# B&R Automation Studio project Parker_BMM_ST_V5_3147_V12 (part 18)

#### cur_save.c
```c
/********************************************************************
 * COPYRIGHT --  B&R CHINA
 ********************************************************************
 * Program: cur_save
 * File: cur_save.c
 * Author: lijianjun
 * Created: March 06, 2013
 ********************************************************************
 * Implementation of program cur_save --- thick profile curve data save/load
 ********************************************************************/

#include <bur/plctypes.h>
#include <string.h>

#ifdef _DEFAULT_INCLUDES
#include <AsDefault.h>
#endif

/***********************************************************************************
**                            Include user files								  **
***********************************************************************************/
#include "draw.h"
#include "recipe.h"
#include "keyap2100.h"
#include "pic_id.h"

/***********************************************************************************
** 					 	       Macro Define								          **
***********************************************************************************/
#define  S$CURVE_NUM	5

#define S$STEP_INIT_OK  10000

#define S$STEP_IDLE     100
#define S$STEP_READ     1000
#define S$STEP_WRITE    2000

#define S$STEP_ERROR	   30000

#define S$WAIT_COMMAND			   0

#define S$ROOT_DISK_SAVE		   100
#define S$ROOT_DISK_LOAD		   200
#define S$ROOT_DISK_CLEAR		   500

#define S$USB_SINGLE_OPEN_SAVE	1000
#define S$USB_SINGLE_CREATE		1100
#define S$USB_SINGLE_WRITE		   1300

#define S$USB_SINGLE_OPEN_LOAD	2000
#define S$USB_SINGLE_READ_MEM	   2100
#define S$USB_SINGLE_READ			2200

#define S$USB_SINGLE_CLOSE		   3000

#define S$USB_ALL_OPEN_SAVE	   11000
#define S$USB_ALL_CREATE		   11100
#define S$USB_ALL_MEM_ALLOC	   11200
#define S$USB_ALL_MEM_GET	      11300
#define S$USB_ALL_WRITE		      11400
#define S$USB_ALL_MEM_FREE		   11500

#define S$USB_ALL_OPEN_LOAD	   12000
#define S$USB_ALL_ALLOC_MEM	   12100
#define S$USB_ALL_READ			   12200
#define S$USB_ALL_READ_WRITE	   12300
#define S$USB_ALL_FREE_MEM  	   12400

#define S$USB_ALL_CLOSE		      13000

#define S$ERROR_STEP			      40000
/**********************************************************************************
**                          Function Declarations								 **
**********************************************************************************/
void changeCurve(USINT *enable);
void newCurve();
void writeData(UINT Index);
void readData(UINT Index);
void initCurve(unsigned short length);
/**********************************************************************************
**     	        		I N I T U P  O F   T H E   T A S K 		 				 **
**********************************************************************************/
_INIT  void init(void)
{
	strcpy(fileSingleName, "curve.usb");		/* file single name */
	strcpy(fileAllName, "curveAll.usb");		/* file all name */

	strcpy(DataObjOperate.ModName,"recCurve");
	strcpy(DataObjOperate.Status,"");
	DataObjOperate.InitStep = 100;
}/*end of INIT*/

/**********************************************************************************
**        			C Y C L I C   P A R T   O F   T H E   T A S K  				 **
**********************************************************************************/
_CYCLIC void cyc(void)
{
	/*  配方名字及数据初始化  */
	switch(DataObjOperate.InitStep)
	{
		case 100:
			/* Initialize info structure */
			DataObjOperate.Ident = 0;
			DatObj_Info.enable	= 1;
			DatObj_Info.pName	   = (UDINT)DataObjOperate.ModName;

			/* Call  FUB  */
			DatObjInfo(&DatObj_Info);

			if(doERR_MODULNOTFOUND == DatObj_Info.status)
			{
				DatObj_Info.enable = 0;
				DataObjOperate.InitStep = 200;
			}
			else if(0 == DatObj_Info.status)
			{
				DatObj_Info.enable = 0;
				DataObjOperate.Ident = DatObj_Info.ident;
				DataObjOperate.InitStep  = 500;
			}
			else if (DatObj_Info.status != ERR_FUB_BUSY)
			{
				DatObj_Info.enable = 0;
				DataObjOperate.InitStep = 40000;
			}
			break;

		case 200:
			/* Initialize create structure */
			DatObj_Create.enable = 1;
			DatObj_Create.grp	 	= 0;
			DatObj_Create.pName 	= (UDINT)DataObjOperate.ModName;
			DatObj_Create.len 	= sizeof(curveData)*(S$NUM_RECIPE + 1);
				DatObj_Create.MemType  = doUSRROM;
			DatObj_Create.Option   = 0;
			DatObj_Create.pCpyData = 0;

			/* Call FUB */
			DatObjCreate(&DatObj_Create);

			if(0 == DatObj_Create.status)
			{
				DataObjOperate.Ident = DatObj_Create.ident;
				DataObjOperate.InitStep = 300;
			}
			break;

		case 300:
			counter = 0;
			initCurve(S$THICK_INIT_LENGTH);
				DataObjOperate.InitStep = 350;
			break;

		case 350:
			status_tmpalloc = TMP_alloc(sizeof(curveData) * (S$NUM_RECIPE + 1), (void*)&pCurveData);
				if(0 == status_tmpalloc)
			{
				for(i=0;i<(S$NUM_RECIPE+1) * S$CURVE_NUM;i++)
					{
					((curveData_typ *)pCurveData)[i] = curveData[0];
				}
				DataObjOperate.InitStep = 380;
			}
			else
			{
				DataObjOperate.InitStep = 40001;
			}
			break;

		case 380:
			DatObj_Write.enable  = 1;
			DatObj_Write.ident 	= DataObjOperate.Ident;
			DatObj_Write.Offset  = 0;
			DatObj_Write.pSource = (UDINT)pCurveData;
			DatObj_Write.len 	   = sizeof(curveData) * (S$NUM_RECIPE + 1);

				/* Call FUB */
				DatObjWrite(&DatObj_Write);

			if(0 == DatObj_Write.status )
			{
				DataObjOperate.InitStep = 400;
			}
			break;

		case 400:
			status_tmpfree = TMP_free(sizeof(curveData) * (S$NUM_RECIPE + 1), (void*)pCurveData);
				if(0 == status_tmpfree)
			{
				readData(curveIndex);
				DataObjOperate.InitStep = 700;
			}
			else
			{
				DataObjOperate.InitStep = 40002;
			}
			break;

		case 500:
			if(1 == gRecipeOperate.NameOk)
			{
				DataObjOperate.InitStep = 600;
			}
			break;

		case 600:
			/* Initialize read structure */
			DatObj_Read.enable 		 = 1;
			DatObj_Read.ident 		 = DataObjOperate.Ident;
			DatObj_Read.Offset 		 = sizeof(curveData) * S$NUM_RECIPE;
			DatObj_Read.pDestination = (UDINT) &curveData;
			DatObj_Read.len 		    = sizeof (curveData);

			/* Call FUB */
			DatObjRead(&DatObj_Read);
			if (curveData[0].usedIndex < S$CURVE_NUM )
				{
				curveIndex = curveData[0].usedIndex;
			}
			else
			{
				curveIndex	= S$CURVE_NUM - 1;
			}

			readData(curveIndex);

			if(0 == DatObj_Read.status)
			{
				DataObjOperate.InitStep = 700;
			}
			else
			{
				DataObjOperate.InitStep = S$STEP_ERROR;
			}
			break;

		case 700:       /*   recipe data  ok*/
			gRecipeOperate.CurveOk  = 1;
			strcpy(DataObjOperate.Status,"curvedata init ok !");
			DataObjOperate.Step     = S$STEP_IDLE;
			DataObjOperate.InitStep = S$STEP_INIT_OK;
			break;

		case S$STEP_INIT_OK:
				break;

		case S$STEP_ERROR:
				break;

		default:
			break;
	}/* switch(DataObjOperate.InitStep) */

	if((0 == DataObjOperate.Ident)||(DataObjOperate.InitStep != S$STEP_INIT_OK ))
		{
		gRecipeOperate.CurveUSBSave = 0;
		gRecipeOperate.CurveUSBLoad = 0;
		curveIndexOld = curveIndex;
		return;
	}

	/* ----------------- Step machine control ----------------- */
	switch (DataObjOperate.Step)
	{
		case S$WAIT_COMMAND:
				gRecipeOperate.usbCurveOk = 1;
			if(1 == gRecipeOperate.CurveSave)
			{
				gRecipeOperate.CurveSave = 0;
				indexRecipe = S$NUM_RECIPE;			/*  current recipe in data module-index = S$NUM_RECIPE */
				DataObjOperate.Step = S$ROOT_DISK_SAVE;
			}/* else if(1 == gRecipeOperate.CurveSave) */
			else if(1 == gRecipeOperate.CurveLoad)
			{
				gRecipeOperate.CurveLoad = 0;
				indexRecipe = S$NUM_RECIPE;			/*  current recipe in data module-index = S$NUM_RECIPE */
				DataObjOperate.Step = S$ROOT_DISK_LOAD;
			}/* else if(1 == gRecipeOperate.CurveSave) */
			else if(1 == gRecipeOperate.CurveRecipeSave)
			{
				gRecipeOperate.CurveRecipeSave = 0;
				indexRecipe = gRecipeOperate.Index % S$NUM_RECIPE;
				DataObjOperate.Step = S$ROOT_DISK_SAVE;
			}/* else if(1 == gRecipeOperate.CurveSave) */
			else if(1 == gRecipeOperate.CurveRecipeLoad)
			{
				gRecipeOperate.CurveRecipeLoad = 0;
				indexRecipe = gRecipeOperate.Index % S$NUM_RECIPE;
				DataObjOperate.Step = S$ROOT_DISK_LOAD;
				gRecipeOperate.CurveSave = 1;		/*  read from recipe then write to current recipe(S$NUM_RECIPE) in data module */
			}/* else if(1 == gRecipeOperate.CurveSave) */
			else if(1 == gRecipeOperate.CurveUSBSave)
			{
				gRecipeOperate.usbCurveOk = 0;
				gRecipeOperate.CurveUSBSave = 0;
				DataObjOperate.Step = S$USB_SINGLE_OPEN_SAVE;
			}/* else if(1 == gRecipeOperate.CurveUSBSave) */
			else if(1 == gRecipeOperate.CurveUSBLoad)
			{
				gRecipeOperate.usbCurveOk = 0;
				gRecipeOperate.CurveUSBLoad = 0;
				DataObjOperate.Step = S$USB_SINGLE_OPEN_LOAD;
				gRecipeOperate.CurveSave = 1;		/*  read from USB then write to current recipe(S$NUM_RECIPE) in data module */
			}/* else if(1 == gRecipeOperate.CurveUSBLoad) */
			else if(1 == gRecipeOperate.CurveUSBLoadAll)
			{
				gRecipeOperate.usbCurveOk = 0;
				gRecipeOperate.CurveUSBLoadAll = 0;
				DataObjOperate.Step = S$USB_ALL_OPEN_LOAD;
			}
			else if(1 == gRecipeOperate.CurveUSBSaveAll)
			{
				gRecipeOperate.usbCurveOk = 0;
				gRecipeOperate.CurveUSBSaveAll = 0;
				DataObjOperate.Step = S$USB_ALL_OPEN_SAVE;
			}
			break;

		/* ---------------- Save to root disk ---------------- */
		case S$ROOT_DISK_SAVE:
				curveData[0].usedIndex = curveIndex;
			writeData(curveIndex);
			/* Initialize write structure */
			DatObj_Write.enable 	= 1;
			DatObj_Write.ident 	= DataObjOperate.Ident;
			DatObj_Write.Offset 	= sizeof(curveData)*indexRecipe;
			DatObj_Write.pSource = (UDINT)&curveData;
			DatObj_Write.len 	   = sizeof(curveData);

			/* Call FUB */
			DatObjWrite(&DatObj_Write);

			if(DatObj_Write.status == 0)
			{
				strcpy(DataObjOperate.Status,"curvedata write ok !");
			}
			else
			{
				strcpy(DataObjOperate.Status,"curvedata write false !");
			}

			DataObjOperate.Step = S$WAIT_COMMAND;
			break;

		/* ---------------- Load from root disk ---------------- */
		case S$ROOT_DISK_LOAD:
				/* Initialize read structure */
				DatObj_Read.enable 		  = 1;
			DatObj_Read.ident 		  = DataObjOperate.Ident;
			DatObj_Read.Offset 		  = sizeof(curveData)*indexRecipe;
			DatObj_Read.pDestination  = (UDINT)&curveData;
			DatObj_Read.len 		     = sizeof(curveData);

			/* Call FUB */
			DatObjRead(&DatObj_Read);

			if(DatObj_Read.status == 0)
			{
				strcpy(DataObjOperate.Status,"curvedata read ok !");
			}
			else
			{
				strcpy(DataObjOperate.Status,"curvedata read false !");
			}

			if (curveData[0].usedIndex < S$CURVE_NUM)
				{
				curveIndex = curveData[0].usedIndex;
			}
			else
			{
				curveIndex	= S$CURVE_NUM - 1;
			}

			readData(curveIndex);

			DataObjOperate.Step = S$WAIT_COMMAND;
			break;

		/* --------------------------------------------------------------- */
		/* ---------------- Save Single curve to usb disk ---------------- */
		/* --------------------------------------------------------------- */
		case S$USB_SINGLE_OPEN_SAVE:			/* file OPEN for save  */
				FileOpen_0.enable  = 1;
			FileOpen_0.pDevice = (UDINT)&gRecipeOperate.deviceNameUSB;
			FileOpen_0.pFile   = (UDINT)&fileSingleName;
			FileOpen_0.mode    = fiREAD_WRITE;

			/* Call FUB */
			FileOpen(&FileOpen_0);

			if(fiERR_FILE_NOT_FOUND == FileOpen_0.status)/* no file   */
			{
				FileOpen_0.enable  = 0;
				DataObjOperate.Step = S$USB_SINGLE_CREATE;
			}
			else
			{
				if(ERR_OK == FileOpen_0.status)			/* file exist */
				{
					FileOpen_0.enable  = 0;
					if(FileOpen_0.filelen == sizeof(curveData))
					{
						DataObjOperate.IdentUSB = FileOpen_0.ident;
						DataObjOperate.Step = S$USB_SINGLE_WRITE;
					}
					else
					{
						gImply.CurveUSB_Length = 1;
						DataObjOperate.Step = S$USB_SINGLE_CLOSE;
					}
				}
				else if (FileOpen_0.status != ERR_FUB_BUSY)
				{
					FileOpen_0.enable  = 0;
					gImply.CurveOP_False = 1;
					DataObjOperate.Step = S$ERROR_STEP;
				}
			}
			break;

		case S$USB_SINGLE_CREATE:			/* file not exist, create*/
				FileCreate_0.enable  = 1;
			FileCreate_0.pDevice = (UDINT)&gRecipeOperate.deviceNameUSB;
			FileCreate_0.pFile   = (UDINT)&fileSingleName;

			/* Call FUB */
			FileCreate(&FileCreate_0);

			if(ERR_OK == FileCreate_0.status)		/* ok */
			{
				FileCreate_0.enable = 0;
				DataObjOperate.IdentUSB = FileCreate_0.ident;
				DataObjOperate.Step = S$USB_SINGLE_WRITE;
			}
			else if (FileCreate_0.status != ERR_FUB_BUSY)
			{
				FileCreate_0.enable= 0;
				gImply.CurveOP_False = 1;
				DataObjOperate.Step = S$USB_SINGLE_CLOSE;
			}
			break;

		case S$USB_SINGLE_WRITE:		/* file write */
				FileWrite_0.enable = 1;
			FileWrite_0.ident  = DataObjOperate.IdentUSB;
			FileWrite_0.offset = 0;
			FileWrite_0.pSrc = (UDINT)&curveData;
			FileWrite_0.len  = sizeof(curveData);

			/* Call FUB */
			FileWrite(&FileWrite_0);

			if(ERR_OK == FileWrite_0.status)				/* ok */
			{
				FileWrite_0.enable = 0;
				gImply.CurveOP_OK = 1;
				DataObjOperate.Step = S$USB_SINGLE_CLOSE;
			}
			else if (FileWrite_0.status != ERR_FUB_BUSY)
			{
				FileWrite_0.enable = 0;
				gImply.CurveOP_False = 1;
				DataObjOperate.Step = S$USB_SINGLE_CLOSE;
			}
			break;

		/* ----------------------------------------------------------------- */
		/* ---------------- Load single curve from USB disk ---------------- */
		/* ----------------------------------------------------------------- */
		case S$USB_SINGLE_OPEN_LOAD:			/* file OPEN  for load  */
				FileOpen_0.enable  = 1;
			FileOpen_0.pDevice = (UDINT)&gRecipeOperate.deviceNameUSB;
			FileOpen_0.pFile   = (UDINT)&fileSingleName;
			FileOpen_0.mode    = fiREAD_WRITE;

			/* Call FUB */
			FileOpen(&FileOpen_0);

			if(fiERR_FILE_NOT_FOUND == FileOpen_0.status)	/* no file   */
			{
				FileOpen_0.enable  = 0;
				gImply.FixUSB_NoFile = 1;
				DataObjOperate.Step = S$WAIT_COMMAND;
			}
			else
			{
				if(ERR_OK == FileOpen_0.status)				/* file exist */
				{
					FileOpen_0.enable = 0;
					if(FileOpen_0.filelen == sizeof(curveData))
					{
						DataObjOperate.IdentUSB = FileOpen_0.ident;
						DataObjOperate.Step = S$USB_SINGLE_READ;
					}
					else
					{
						gImply.CurveUSB_Length = 1;
						DataObjOperate.Step = S$USB_SINGLE_CLOSE;
					}
				}
				else if (FileOpen_0.status != ERR_FUB_BUSY)
				{
					FileOpen_0.enable = 0;
					gImply.CurveOP_False = 1;
					DataObjOperate.Step = S$ERROR_STEP;
				}
			}
			break;

		case S$USB_SINGLE_READ:			/* file single read  */
				FileRead_0.enable = 1;
			FileRead_0.ident  = DataObjOperate.IdentUSB;
			FileRead_0.offset = 0;
			FileRead_0.pDest  = (UDINT)&curveData;
			FileRead_0.len    = sizeof(curveData);

			/* Call FUB */
			FileRead(&FileRead_0);

			if(ERR_OK == FileRead_0.status)	/* ok */
			{
				FileRead_0.enable = 0;
				gImply.CurveOP_OK = 1;
				if (curveData[0].usedIndex < S$CURVE_NUM)
					{
					curveIndex = curveData[0].usedIndex;
				}
				else
				{
					curveIndex	= S$CURVE_NUM - 1;
				}

				readData(curveIndex);

				gRecipeOperate.CurveSave = 1;		/*  read from USB then write to current recipe(S$NUM_RECIPE) in data module */
				DataObjOperate.Step = S$USB_SINGLE_CLOSE;
			}
			else if (FileRead_0.status != ERR_FUB_BUSY)
			{
				FileRead_0.enable = 0;
				gImply.CurveOP_False = 1;
				DataObjOperate.Step = S$USB_SINGLE_CLOSE;
			}
			break;

		/* ------------------------------------------------------- */
		/* ---------------- Close USB file device ---------------- */
		/* ------------------------------------------------------- */
		case S$USB_SINGLE_CLOSE:			/* file close*/
				FileClose_0.enable = 1;
			FileClose_0.ident  = DataObjOperate.IdentUSB;

			/* Call FBK */
			FileClose(&FileClose_0);

			if(ERR_OK == FileClose_0.status)	/* ok */
			{
				FileClose_0.enable = 0;
				DataObjOperate.Step = S$WAIT_COMMAND;
			}
			else if (FileClose_0.status != ERR_FUB_BUSY)
			{
				FileClose_0.enable = 0;
				DataObjOperate.Step = S$ERROR_STEP;
			}
			break;

		/* ------------------------------------------------------ */
		/* ---------------- All Save to usb disk ---------------- */
		/* ------------------------------------------------------ */
		case S$USB_ALL_OPEN_SAVE:			/* file OPEN for save  */
				FileOpen_0.enable  = 1;
			FileOpen_0.pDevice = (UDINT)&gRecipeOperate.deviceNameUSB;
			FileOpen_0.pFile   = (UDINT)&fileAllName;
			FileOpen_0.mode    = fiREAD_WRITE;

			/* Call FUB */
			FileOpen(&FileOpen_0);

			if(fiERR_FILE_NOT_FOUND == FileOpen_0.status)/* no file   */
			{
				FileOpen_0.enable   = 0;
				DataObjOperate.Step = S$USB_ALL_CREATE;
			}
			else
			{
				if(ERR_OK == FileOpen_0.status)			/* file exist */
				{
					FileOpen_0.enable  = 0;
					if(FileOpen_0.filelen == sizeof(curveData)*(S$NUM_RECIPE + 1))
						{
						DataObjOperate.IdentAllUSB = FileOpen_0.ident;
						DataObjOperate.Step = S$USB_ALL_MEM_ALLOC;
					}
					else
					{
						gImply.CurveUSB_Length = 1;
						DataObjOperate.Step = S$USB_ALL_CLOSE;
					}
				}
				else if (FileOpen_0.status != ERR_FUB_BUSY)
				{
					FileOpen_0.enable  = 0;
					gImply.CurveOP_False = 1;
					DataObjOperate.Step = S$ERROR_STEP;
				}
			}
			break;

		case S$USB_ALL_CREATE:			/* file not exist, create*/
				FileCreate_0.enable  = 1;
			FileCreate_0.pDevice = (UDINT)&gRecipeOperate.deviceNameUSB;
			FileCreate_0.pFile   = (UDINT)&fileAllName;

			/* Call FUB */
			FileCreate(&FileCreate_0);

			if(ERR_OK == FileCreate_0.status)		/* ok */
			{
				FileCreate_0.enable = 0;
				DataObjOperate.IdentAllUSB = FileCreate_0.ident;
				DataObjOperate.Step = S$USB_ALL_MEM_ALLOC;
			}
			else if (FileCreate_0.status != ERR_FUB_BUSY)
			{
				FileCreate_0.enable = 0;
				gImply.CurveOP_False = 1;
				DataObjOperate.Step = S$USB_ALL_CLOSE;
			}
			break;

		case S$USB_ALL_MEM_ALLOC:	/* file request All memory */
				status_tmpalloc = TMP_alloc(sizeof(curveData)*(S$NUM_RECIPE + 1), (void*)&pCurveData);
				if(0 == status_tmpalloc)
			{
				memset((void *)pCurveData,0,sizeof(curveData)*(S$NUM_RECIPE + 1));
					DataObjOperate.Step = S$USB_ALL_MEM_GET;
			}
			else
			{
				gImply.CurveOP_False = 1;
				DataObjOperate.Step = S$USB_ALL_CLOSE;
			}
			break;

		case S$USB_ALL_MEM_GET:
				DatObj_Read.enable = 1;
			DatObj_Read.ident  = DataObjOperate.Ident;
			DatObj_Read.Offset = 0;
			DatObj_Read.pDestination = (UDINT)pCurveData;
			DatObj_Read.len = sizeof(curveData)*(S$NUM_RECIPE + 1);

				/* Call FUB */
				DatObjRead(&DatObj_Read);
			if(0 == DatObj_Read.status)
			{
				DatObj_Read.enable = 0;
				DataObjOperate.Step = S$USB_ALL_WRITE;
			}
			else if (DatObj_Read.status != ERR_FUB_BUSY)
			{
				DatObj_Read.enable = 0;
				gImply.CurveOP_False = 1;
				DataObjOperate.Step = S$USB_ALL_MEM_FREE;
			}
			break;

		case S$USB_ALL_WRITE:		/* file single write */
				FileWrite_0.enable = 1;
			FileWrite_0.ident  = DataObjOperate.IdentAllUSB;
			FileWrite_0.offset = 0;
			FileWrite_0.pSrc = (UDINT)pCurveData;
			FileWrite_0.len  = sizeof(curveData)*(S$NUM_RECIPE + 1);

				/* Call FUB */
				FileWrite(&FileWrite_0);

			if(ERR_OK == FileWrite_0.status)				/* ok */
			{
				FileWrite_0.enable = 0;
				gImply.CurveOP_OK = 1;
				DataObjOperate.Step = S$USB_ALL_MEM_FREE;
			}
			else if (FileWrite_0.status != ERR_FUB_BUSY)
			{
				FileWrite_0.enable = 0;
				gImply.CurveOP_False = 1;
				DataObjOperate.Step = S$USB_ALL_MEM_FREE;
			}
			break;

		case S$USB_ALL_MEM_FREE:
				status_tmpfree = TMP_free(sizeof(curveData)*(S$NUM_RECIPE + 1), (void*)pCurveData);
				if(0 == status_tmpfree)
			{
				DataObjOperate.Step = S$USB_ALL_CLOSE;
			}
			else
			{
				DataObjOperate.Step = S$USB_ALL_CLOSE;
			}
			break;

		/* ----------------------------------------------------------- */
		/* ----------------  All Load from USB disk   ---------------- */
		/* ----------------------------------------------------------- */
		case S$USB_ALL_OPEN_LOAD:			/* file OPEN  for load  */
				FileOpen_0.enable  = 1;
			FileOpen_0.pDevice = (UDINT)&gRecipeOperate.deviceNameUSB;
			FileOpen_0.pFile   = (UDINT)&fileAllName;
			FileOpen_0.mode    = fiREAD_WRITE;

			/* Call FUB */
			FileOpen(&FileOpen_0);

			if(fiERR_FILE_NOT_FOUND == FileOpen_0.status)	/* no file   */
			{
				FileOpen_0.enable  = 0;
				gImply.CurveUSB_NoFile = 1;
				DataObjOperate.Step = S$WAIT_COMMAND;
			}
			else
			{
				if(ERR_OK == FileOpen_0.status)				/* file exist */
				{
					FileOpen_0.enable = 0;
					if(FileOpen_0.filelen == sizeof(curveData)*(S$NUM_RECIPE + 1))
						{
						DataObjOperate.IdentAllUSB = FileOpen_0.ident;
						DataObjOperate.Step = S$USB_ALL_ALLOC_MEM;
					}
					else
					{
						gImply.CurveUSB_Length = 1;
						DataObjOperate.Step = S$USB_ALL_CLOSE;
					}
				}
				else if (FileOpen_0.status != ERR_FUB_BUSY)
				{
					FileOpen_0.enable = 0;
					gImply.CurveOP_False = 1;
					DataObjOperate.Step = S$ERROR_STEP;
				}
			}
			break;

		case S$USB_ALL_ALLOC_MEM:			/* file  read request memory */
				status_tmpalloc = TMP_alloc(sizeof(curveData)*(S$NUM_RECIPE + 1), (void*)&pCurveData);
				if(0 == status_tmpalloc)
			{
				DataObjOperate.Step = S$USB_ALL_READ;
			}
			else
			{
				gImply.CurveOP_False = 1;
				DataObjOperate.Step = S$USB_ALL_CLOSE;
			}
			break;

		case S$USB_ALL_READ:			/* file  read  */
				FileRead_0.enable = 1;
			FileRead_0.ident  = DataObjOperate.IdentAllUSB;
			FileRead_0.offset = 0;
			FileRead_0.pDest  = (UDINT)pCurveData;
			FileRead_0.len    = sizeof(curveData)*(S$NUM_RECIPE + 1);

				/* Call FUB */
				FileRead(&FileRead_0);

			if(ERR_OK == FileRead_0.status)	/* ok */
			{
				FileRead_0.enable = 0;
				DataObjOperate.Step = S$USB_ALL_READ_WRITE;
			}
			else if (FileRead_0.status != ERR_FUB_BUSY)
			{
				FileRead_0.enable = 0;
				gImply.CurveOP_False = 1;
				DataObjOperate.Step = S$USB_ALL_FREE_MEM;
			}
			break;

		case S$USB_ALL_READ_WRITE:
				DatObj_Write.enable  = 1;
			DatObj_Write.ident 	 = DataObjOperate.Ident;
			DatObj_Write.Offset  = 0;
			DatObj_Write.pSource = (UDINT)pCurveData;
			DatObj_Write.len 	 = sizeof(curveData)*(S$NUM_RECIPE + 1);

				DatObjWrite(&DatObj_Write);

			if(0 == DatObj_Write.status)
			{
				DatObj_Write.enable  = 0;
				gImply.CurveOP_OK = 1;
				gRecipeOperate.CurveLoad = 1;
				DataObjOperate.Step = S$USB_ALL_FREE_MEM;
			}
			else if (DatObj_Write.status != ERR_FUB_BUSY)
			{
				DatObj_Write.enable  = 0;
				gImply.CurveOP_False = 1;
				DataObjOperate.Step = S$USB_ALL_FREE_MEM;
			}
			break;

		case S$USB_ALL_FREE_MEM:
				status_tmpfree = TMP_free(sizeof(curveData)*(S$NUM_RECIPE + 1), (void*)pCurveData);
				if(0 == status_tmpfree)
			{
				DataObjOperate.Step = S$USB_ALL_CLOSE;
			}
			else
			{
				DataObjOperate.Step = S$USB_ALL_CLOSE;
			}
			break;
		/* ----------------------------------------------------------- */
		/* ---------------- All Close USB file device ---------------- */
		/* ----------------------------------------------------------- */
		case S$USB_ALL_CLOSE:			/* file close*/
				FileClose_0.enable = 1;
			FileClose_0.ident  = DataObjOperate.IdentAllUSB;

			/* Call FBK */
			FileClose(&FileClose_0);

			if(ERR_OK == FileClose_0.status)	/* ok */
			{
				FileClose_0.enable = 0;
				DataObjOperate.Step = S$WAIT_COMMAND;
			}
			else if (FileClose_0.status != ERR_FUB_BUSY)
			{
				FileClose_0.enable = 0;
				DataObjOperate.Step = S$ERROR_STEP;
			}
			break;

		case S$ERROR_STEP:
				DataObjOperate.Step = S$WAIT_COMMAND;
			break;
	}/* switch (DataObjOperate.Step) */

	if(1 == bCurveIndexChgBtn)
	{
		bCurveIndexChgBtn = 0;
		curveIndex = curveIndex + 1;
		curveIndex = curveIndex % 5;
	}

	if(curveIndex != curveIndexOld)
	{
		ChangeEnable = 1;
		changeCurve(&ChangeEnable);
		bCurveIndexChange = 1;
	}
	curveIndexOld = curveIndex;

}/*end of CYCLIC*/

/**************************************************************************************
**        				FUNCTION  REALIZE				   							 **
**************************************************************************************/
void changeCurve(USINT *enable)
{

	if (1 == *enable)
	{
		writeData(curveIndexOld);

		/*curveIndex = curveIndex + 1;*/

		curveIndex = curveIndex % S$CURVE_NUM;

		if (curveData[curveIndex].CurveNode[S$THICK_MAX].v3.y == 0)
			{
			newCurve();
		}
		else
		{
			readData(curveIndex);
		}

		*enable = 0;
	}
}

void newCurve()
{
	memset(SetPos,0,sizeof(SetPos));
	memset(CurveNode,0,sizeof(CurveNode));

	for( i = 0; i<= S$THICK_MAX; i++)
		{
		DrawMan.weight = 300;
		SetPos[i].x = DrawMan.weight;
		SetPos[i].y = i;
	}

	DrawMan.oldWeight 			=  DrawMan.weight;
	DrawMan.v1 						=  (DrawMan.weight) + 1;
	DrawMan.v2 						=  (DrawMan.weight) + 1;
	DrawMan.v03 					=  0;
	DrawMan.currentNode  		=  S$THICK_MAX;
	DrawMan.currentPoint 		=  0;
	DrawMan.flagLineFocus 		=  0;
	CurveNode[0].former    	=  S$THICK_MAX;
	CurveNode[0].next    		=  S$THICK_MAX;
	CurveNode[0].v3.x    		=  DrawMan.weight;
	CurveNode[0].v3.y    		=  0;
	CurveNode[0].flagNode  		=  1;

	CurveNode[S$THICK_MAX].former 	= 0;
	CurveNode[S$THICK_MAX].next   	= 0;
	CurveNode[S$THICK_MAX].v0.x   	= DrawMan.weight;
	CurveNode[S$THICK_MAX].v0.y   	= 0;
	CurveNode[S$THICK_MAX].v3.x   	= DrawMan.weight;
	CurveNode[S$THICK_MAX].v3.y   	= S$THICK_MAX;

	CurveNode[S$THICK_MAX].v1.x   	= (DrawMan.weight) + 1;
	CurveNode[S$THICK_MAX].v1.y   	= CurveNode[S$THICK_MAX].v0.y +
		(CurveNode[S$THICK_MAX].v3.y - CurveNode[S$THICK_MAX].v0.y)*1/
		3 ;
		CurveNode[S$THICK_MAX].v2.x   	= (DrawMan.weight) + 1;
	CurveNode[S$THICK_MAX].v2.y   	= CurveNode[S$THICK_MAX].v0.y +
		(CurveNode[S$THICK_MAX].v3.y - CurveNode[S$THICK_MAX].v0.y)*(S$THICK_V_SCALE -1)/
		S$THICK_V_SCALE;

	CurveNode[S$THICK_MAX].flagNode =  1;

	setColor = 1;
}/*end of function */

void readData(UINT Index)
{
	Index = Index % 5;
	memcpy(CurveNode,curveData[Index].CurveNode,sizeof(CurveNode));
	memcpy(SetPos,curveData[Index].SetPos,sizeof(SetPos));
	DrawMan.weight 	   = 	curveData[Index].weight;
	DrawMan.oldWeight 	=  DrawMan.weight;
	DrawMan.v1 				= 	curveData[Index].v1;
	DrawMan.v2				= 	curveData[Index].v2;
	DrawMan.v03				= 	curveData[Index].v03;
	DrawMan.currentPoint	=	curveData[Index].currentPoint;
	DrawMan.currentNode	=	curveData[Index].currentNode;
	DrawMan.flagLineFocus=	curveData[Index].flagLineFocus;

}/*end of function */

void writeData(UINT Index)
{
	Index = Index % 5;
	memcpy(curveData[Index].CurveNode,CurveNode,sizeof(CurveNode));
	memcpy(curveData[Index].SetPos,SetPos,sizeof(SetPos));
	curveData[Index].weight 			= 	DrawMan.weight;
	curveData[Index].v1 				   = 	DrawMan.v1;
	curveData[Index].v2			      = 	DrawMan.v2;
	curveData[Index].v03				   = 	DrawMan.v03;
	curveData[Index].currentPoint	   =	DrawMan.currentPoint;
	curveData[Index].currentNode	   =	DrawMan.currentNode;
	curveData[Index].flagLineFocus	=	DrawMan.flagLineFocus;

}/*end of function */
void initCurve(unsigned short length)
{
	memset(curveData[0].SetPos,0,sizeof(curveData[0].SetPos));
	memset(curveData[0].CurveNode,0,sizeof(curveData[0].CurveNode));

	for( i = 0; i<= S$THICK_MAX; i++)
		{
		curveData[0].SetPos[i].x = length;
		curveData[0].SetPos[i].y = i;
	}

	curveData[0].weight        =  0;
	curveData[0].v1 	         =  length+1;
	curveData[0].v2		      =  length+1;
	curveData[0].v03	         =  length;
	curveData[0].currentNode   =  S$THICK_MAX;
	curveData[0].currentPoint  =  0;
	curveData[0].flagLineFocus =  0;
	curveData[0].usedIndex     =  0;

	curveData[0].CurveNode[0].former   =  S$THICK_MAX;
	curveData[0].CurveNode[0].next     =  S$THICK_MAX;
	curveData[0].CurveNode[0].v3.x     =  length;
	curveData[0].CurveNode[0].v3.y     =  0;
	curveData[0].CurveNode[0].flagNode  =  1;

	curveData[0].CurveNode[S$THICK_MAX].former 	= 0;
	curveData[0].CurveNode[S$THICK_MAX].next   	= 0;
	curveData[0].CurveNode[S$THICK_MAX].v0.x   	= length;
	curveData[0].CurveNode[S$THICK_MAX].v0.y   	= 0;
	curveData[0].CurveNode[S$THICK_MAX].v3.x   	= length;
	curveData[0].CurveNode[S$THICK_MAX].v3.y   	= S$THICK_MAX;

	curveData[0].CurveNode[S$THICK_MAX].v1.x   	= length+1;
	curveData[0].CurveNode[S$THICK_MAX].v1.y   	= CurveNode[S$THICK_MAX].v0.y +
		(curveData[0].CurveNode[S$THICK_MAX].v3.y - curveData[0].CurveNode[S$THICK_MAX].v0.y)*1/3 ;
		curveData[0].CurveNode[S$THICK_MAX].v2.x   	= length+1;
	curveData[0].CurveNode[S$THICK_MAX].v2.y   	= CurveNode[S$THICK_MAX].v0.y +
		(curveData[0].CurveNode[S$THICK_MAX].v3.y - curveData[0].CurveNode[S$THICK_MAX].v0.y)*2/3;
		curveData[0].CurveNode[S$THICK_MAX].flagNode =  1;

	memcpy(&curveData[1],&curveData[0],sizeof(curveData_typ));
	memcpy(&curveData[2],&curveData[0],sizeof(curveData_typ));
	memcpy(&curveData[3],&curveData[0],sizeof(curveData_typ));
	memcpy(&curveData[4],&curveData[0],sizeof(curveData_typ));
}

/*************************************************************************************/
```

### Program Logical/thickness/cur_cal (ANSIC, version 1.00.0) - profile point value

#### cur_cal.c
```c
/**************************************************************************************
 * COPYRIGHT --  B&R CHINA
 **************************************************************************************
 * Program: cur_cal
 * File: cur_cal.c
 * Author: lijianjun
 * Created: March 06, 2013
 *************************************************************************************
 * Implementation of program cur_cal --- thick profile curve data calculation
 ************************************************************************************/

#include <bur/plctypes.h>
#include <string.h>

#ifdef _DEFAULT_INCLUDES
#include <AsDefault.h>
#endif

/***********************************************************************************
** 					 	           Include user files								          **
***********************************************************************************/
#include "draw.h"

/**********************************************************************************
**                             Function Declarations								      **
**********************************************************************************/
void BesselCal(short nodeNum);

/**********************************************************************************
**     	        		      I N I T U P  O F   T H E   T A S K 		 				   **
**********************************************************************************/
_INIT void init ( void )
{
	calStep = 0;
}

/**********************************************************************************
**        			 C Y C L I C   P A R T   O F   T H E   T A S K  				   **
**********************************************************************************/
_CYCLIC void cyclic ( void )
{
	if (oldV2 != DrawMan.v2   && enable == 0 && calStep == 0)enable = 1;
	if (oldV1 != DrawMan.v1   && enable == 0 && calStep == 0)enable = 1;
	if (oldV03 != DrawMan.v03 && enable == 0 && calStep == 0)enable = 1;

	SetPos[0].x  = CurveNode[0].v3.x;
	SetPos[0].y  = 0;
	SetPos[S$THICK_MAX].x = CurveNode[S$THICK_MAX].v3.x;
	SetPos[S$THICK_MAX].y = S$THICK_MAX;

	BesselCal(DrawMan.currentNode);

}/*end of CYCLIC*/

/**************************************************************************************
**        				          FUNCTION  REALIZE				   							 **
**************************************************************************************/
void BesselCal(short nodeNum)
{
	switch (calStep)
	{
		case 0:
			if (1 == enable)
			{
				p0 = &CurveNode[nodeNum];
				p1 = &CurveNode[CurveNode[nodeNum].next];

				v1  = DrawMan.v1;
				v2  = DrawMan.v2;
				v03 = DrawMan.v03;
				if ((p0->v3.y - p0->v0.y) != 0) interval0	= 1/(float)(p0->v3.y - p0->v0.y);
				if ((p1->v3.y - p1->v0.y) != 0) interval1	= 1/(float)(p1->v3.y - p1->v0.y);
				calStep = 10;
			}
			break;
		case 10:
			if (1 == enable)
			{
				if (0 == DrawMan.flagLineFocus)
				{
					p0->v1.x = v1;
					p0->v2.x = v2;
				}
				else
				{
					if (v03 >= (DrawMan.weight) && v03 <= S$THICK_X_LENGTH)
						{
						p0->v3.x = v03;
						p1->v0.x = v03;
						p0->v2.x = v2;
						p1->v1.x = v1;
					}
				}
				calStep = 20;
			}
			break;
		case 20:
			t0  = 0;
			t1  = 0;
			memcpy(oldSetPos,SetPos,sizeof(SetPos));
			calStep = 30;
			break;
		case 30:
			for(i = p0->v0.y + 1 ;i < p0->v3.y ;i++)
			{
				oldSetPos[i].x=(short)((1-t0)*(1-t0)*(1-t0)*(float)p0->v0.x
					+3*t0*(1-t0)*(1-t0)*(float)p0->v1.x
					+3*t0*t0*(1-t0)*(float)p0->v2.x
					+t0*t0*t0*(float)p0->v3.x);

				t0	+= interval0;
				if (oldSetPos[i].x > S$THICK_X_LENGTH || oldSetPos[i].x < DrawMan.weight)
					{
					v1  = oldV1;
					v2  = oldV2;
					v03 = oldV03;

					calStep = 10;
					return;
				}
			}

			if (1 == DrawMan.flagLineFocus)
			{
				calStep = 40;
			}
			else
			{
				calStep = 50;
			}
			break;
		case 40:
			for(i = p1->v0.y + 1 ;i < p1->v3.y ;i++)
			{

				oldSetPos[i].x=(short)((1-t1)*(1-t1)*(1-t1)*(float)p1->v0.x
					+3*t1*(1-t1)*(1-t1)*(float)p1->v1.x
					+3*t1*t1*(1-t1)*(float)p1->v2.x
					+t1*t1*t1*(float)p1->v3.x);

				t1	+= interval1;
				if (oldSetPos[i].x > S$THICK_X_LENGTH || oldSetPos[i].x < DrawMan.weight)
					{

					v1  = oldV1;
					v2  = oldV2;
					v03 = oldV03;

					calStep = 10;
					return;
				}
			}
			oldSetPos[p0->v3.y].x = v03;
			calStep = 50;
			break;
		case 50:
			calStep = 0;
			if (enable != 0)
			{
				enable = 0;
				memcpy(SetPos,oldSetPos,sizeof(SetPos));
				DrawMan.v1 	= oldV1   = v1;
				DrawMan.v2 	= oldV2   = v2;
				DrawMan.v03 = oldV03  = v03;
			}
			break;
	}

}/*end of function*/
```

#### cur_cal.var
```iecst
VAR
	oldSetPos : ARRAY[0..399] OF position_typ;
	enable : USINT;
	calStep : UINT;
	oldV1 : INT;
	oldV2 : INT;
	oldV03 : INT;
	v1 : INT;
	v2 : INT;
	v03 : INT;
	interval0 : REAL;
	interval1 : REAL;
	t0 : REAL;
	t1 : REAL;
	i : UINT;
	p0 : REFERENCE TO curveNode_typ;
	p1 : REFERENCE TO curveNode_typ;
END_VAR
```

### Program Logical/thickness/parison (ANSIC, version 1.00.0) - thickness parison controller

#### parison.c
```c
/**********************************************************************************
 * COPYRIGHT --  B&R China
 **********************************************************************************
 * Program: parison
 * File: parison.c
 * Author: lijianjun
 * Created: March 06, 2013
 **********************************************************************************
 * Implementation of program parison --- thickness controller
 *********************************************************************************/

#include <bur/plctypes.h>

#ifdef _DEFAULT_INCLUDES
#include <AsDefault.h>
#endif

#include <string.h>

#include "defines.h"
#include "thick.h"
#include "keyap2100.h"
//#include "keyap880.h"
#include "pic_id.h"
/**********************************************************************************
**                            Function Declarations								      **
**********************************************************************************/
/**********************************************************************************
**     	        		I N I T U P  O F   T H E   T A S K 		 				         **
**********************************************************************************/
_INIT    void init()
{
	RTInfo_Task.enable = 1;
	RTInfo(&RTInfo_Task);

	tTask = RTInfo_Task.cycle_time/1000.0/1000.0;		/*  from us ---> s  */

	TimePid.e0          = 0;
	TimePid.e1          = 0;
	TimePid.e2          = 0;
	TimePid.OutLast     = 0;
	TimePid.Slew        =  300;
	TimePid.OutMax      =  20000;
	TimePid.OutMin      = -20000;
	TimePid.RepairOut   = -80;
	TimePid.KpGain      = 100;
	TimePid.KiGain      = 5;
	TimePid.KdGain      = 20;
	TimePid.Change      = 30;
	TimePid.Wave        = 30;

	AccuPid.e0          = 0;
	AccuPid.e1          = 0;
	AccuPid.e2          = 0;
	AccuPid.OutLast     = 0;
	AccuPid.Slew        =  300;
	AccuPid.OutMax      =  20000;
	AccuPid.OutMin      = -20000;
	AccuPid.RepairOut   = -80;
	AccuPid.KpGain      = 100;
	AccuPid.KiGain      = 5;
	AccuPid.KdGain      = 20;
	AccuPid.Change      = 30;
	AccuPid.Wave        = 30;

	CalibPid.e0         = 0;
	CalibPid.e1         = 0;
	CalibPid.e2         = 0;
	CalibPid.OutLast    = 0;
	CalibPid.Slew       =  300;
	CalibPid.OutMax     =  20000;
	CalibPid.OutMin     = -20000;
	CalibPid.RepairOut  = -80;
	CalibPid.KpGain     = 50;
	CalibPid.KiGain     = 5;
	CalibPid.KdGain     = 20;
	CalibPid.Change     = 30;
	CalibPid.Wave       = 30;

	Wave = 1;
	gControlInfo.ControlStatus = 0;

	TimeCtrlStep  = 100;
	AccuCtrlStep  = 200;
	CalibrateStep = 0;

	TimeCount     = 0;
	MarkerTime    = 0;
	ContolEndTime = 0;
	gThickIO.In.Purge = 0;

	RampCalibSet.Ts = tTask;
	RampCalibSet.Accel = 3000;
	RampCalibSet.Once = 0;
	RampCalibSet.Set  = gServoLinear.Current;

	HydSCurveRamp(&RampCalibSet);

	RampSet.Ts = tTask;
	RampSet.Accel = 3000;
	RampSet.Once = 0;
	RampSet.Set  = gServoLinear.Current;

	HydRampCos(&RampSet);

	/* differentiator for evaluating the actual speed */
	vHydDT2Set.Ts = tTask;	      /* cycle time 0.002s 			    */
	vHydDT2Set.Tv = 1.0; 	      /* derivative time constant [s]   */
	vHydDT2Set.T1 = 5 * tTask; 	/* filter time constant 1 : 0.01s */
	vHydDT2Set.T2 = 5 * tTask; 	/* filter time constant 2 : 0.01s */

	/* differentiator for evaluating the actual speed */
	vHydDT2Act.Ts = tTask;	      /* cycle time 0.002s 			  */
	vHydDT2Act.Tv = 1.0; 	      /* derivative time constant [s]   */
	vHydDT2Act.T1 = 5 * tTask; 	/* filter time constant 1 : 0.01s */
	vHydDT2Act.T2 = 5 * tTask; 	/* filter time constant 2 : 0.01s */

	vSetLimit = 30;
	vActLimit = 30;

	gThickData.Offset = 0;
	gThickProf.FunOption.SealMode = 0;

	gThickProf.FunOption.Servo = 1;

}/*  end of init  */

/**********************************************************************************
**        			C Y C L I C   P A R T   O F   T H E   T A S K  				      **
**********************************************************************************/

_CYCLIC  void cyc()
{

	/*---------Ext Moog Thick signel-------------*/
	if(1 == gMachineFix.Option.bExtParisonCtrl)
	{
		gThickProf.FunOption.Servo = 0;
		if (1 == gMachineInfo.ExtParisonCtrlStart)	/* 外部壁厚触发 */
		{
			gMachineInfo.ExtParisonCtrlStart = 0;
			gMacTimer.ExtParisonCtrlOffDelay.IN = 1;
			gMacTimer.ExtParisonCtrlOffDelay.PT = 100;
			gMachineOut.ExtParisonCtrl = 1;
		}
		if (1 == gMacTimer.ExtParisonCtrlOffDelay.Q)
		{
			gMacTimer.ExtParisonCtrlOffDelay.IN = 0;
			gMachineOut.ExtParisonCtrl = 0;
		}
	}

	/*---------ipis0116-------------------------------------------------------------------*/

	if( 0 == gThickData.CurrentTime)   // Parision Cycle End
	{
		if(1 == RMold.Option.Enable && 1 == LMold.Option.Enable)
		{
			gThickProf.TimSet.CycleTime =gUserPara.ThickTime_TwoMold;
		}
		else
		{
			gThickProf.TimSet.CycleTime = gUserPara.ThickTime_OneMold;
		}
	}
	/*-----------------------------------------------------------------------------------*/

	gThickIO.enable = gThickProf.FunOption.Servo;
	bHideDieGapMoveFrame = !gThickProf.FunOption.bMoveFrame;
	/*-----------------------------------------------------------------------------------*/

	if(gPanelObj.GetPicture == PIC_GAP_CALIBRATE)
	{
		cmdServoUp = gPanelObj.KeyMatric[S$KEYMATRIX_F5];
		cmdServoDn = gPanelObj.KeyMatric[S$KEYMATRIX_F6];
		cmdAutoCalibrate = gPanelObj.KeyMatric[S$KEYMATRIX_F12];
	}
	else
	{
		cmdServoUp = 0;
		cmdServoDn = 0;
		cmdAutoCalibrate = 0;
	}

	TimePid.Wave   = gThickProf.ShareSet.Wave = 10;
	TimePid.Change = gThickProf.ShareSet.Change;
	TimePid.RepairOut = gThickProf.ShareSet.ServoValveComp;

	AccuPid.Wave   = gThickProf.ShareSet.Wave;
	AccuPid.Change = gThickProf.ShareSet.Change;
	AccuPid.RepairOut = gThickProf.ShareSet.ServoValveComp;

	CalibPid.Wave   = gThickProf.ShareSet.Wave;
	CalibPid.Change = gThickProf.ShareSet.Change;
	CalibPid.RepairOut = gThickProf.ShareSet.ServoValveComp;
	CalibPid.Act = gServoLinear.Current;

	gThickData.CurrentPos = gAccuLinear.Current;
	gThickData.ServoAct   = gServoLinear.Current;

	TimePid.KiGain = 6;
	AccuPid.KiGain = 6;
	CalibPid.KiGain= 6;

	if(0 == gMachineOut.ParisonPump)
	{
		TimePid.KiGain = 0;
		AccuPid.KiGain = 0;
		CalibPid.KiGain= 0;
	}

	/* velocity  */
	vHydDT2Act.u = gServoLinear.Current;
	HydDT2(&vHydDT2Act);

	/* velocity  */
	vHydDT2Set.u = SetValue;
	HydDT2(&vHydDT2Set);

	/*  servo LVDT calibration OK or NOT OK  */
	if((gServoLinear.MaxPos  > gServoLinear.ZeroPos + 2000) && (gServoLinear.MaxPos < 32000)&&
		(gServoLinear.ZeroPos > 500))
	{
		gServoLinear.IsReady = 1;
	}
	else
	{
		gServoLinear.IsReady = 0;
	}

	if(0 == CalibrateStep)gServoLinear.Status = gServoLinear.IsReady; /* not auto calibration */

	if(gControlInfo.ControlStatus == S$STATUS_AUTORUN) /* 非调校状态 */
		{
		if(1 == gThickIO.In.StartThick)	/* 壁厚触发 */
		{
			if(0 == gThickProf.FunOption.IsAccu)
			{
				if(gThickData.TimePerDot != 0)TimeCtrlStep = 10;
				AccuCtrlStep = 0;
			}
			else
			{
				TimeCtrlStep = 0;
				AccuCtrlStep = 10;
			}
			StartTime = 250;
			gThickIO.In.StartThick = 0;
		}

		if(1 == gThickIO.In.Stop)       /* 停止信号 */
		{
			if(1 == gThickProf.FunOption.IsAccu)
			{
				AccuCtrlStep = 50;
			}
			gThickIO.In.Stop = 0;
		}

		if(gThickIO.tSealGapDly > 0.0)
		{
			gThickIO.tSealGapDly = gThickIO.tSealGapDly - tTask;
			if(gThickIO.tSealGapDly < 0.0)gThickIO.tSealGapDly = 0.0;
			if(gThickIO.tSealGapDly < 2 * tTask)gThickIO.In.SealGap = 1;
		}

		if(1 == gThickIO.In.SealGap)    /* 封口信号 */
		{
			if(0 == gThickProf.FunOption.IsAccu)
			{
				TimeCtrlStep = 110;
				AccuCtrlStep = 0;
			}
			else
			{
				TimeCtrlStep = 0;
				AccuCtrlStep = 100;
			}
			gThickIO.In.SealGap = 0;
		}

		TimePid.Act = gServoLinear.Current;
		AccuPid.Act = gServoLinear.Current;

		if(0 == gThickProf.FunOption.IsAccu) 	/* 时间式 */
		{
			switch(TimeCtrlStep)
			{
				case 10:
					gThickData.Counter = 0;
					gThickData.StartServoPos = TimePid.Act ;
					TimePid.OutMax =  gThickProf.ShareSet.StartFlow * 33;
					TimePid.OutMin = -1 * TimePid.OutMax ;

					RampSet.Once = 0;
					SetPID = TimePid.Act;

					TimeCtrlStep = 20;
					break;

				case 20:
					gThickData.Counter++;                    				/* 开口延迟 */

					if((gThickData.SetData[0] - gThickData.StartServoPos != 0) && (gThickData.TimeOpenDly != 0))
					{
						SetPID = (short)(gThickData.StartServoPos + (gThickData.SetData[0] - gThickData.StartServoPos)
							* gThickData.Counter / gThickData.TimeOpenDly );
					}
					else
					{
						SetPID = gThickData.SetData[0];
					}

					if(gThickData.Counter > gThickData.TimeOpenDly)
					{
						gThickData.Counter = 0;
						TimeCtrlStep = 30;
					}
					break;

				case 30:
					memset(gThickData.RealData ,0,sizeof(gThickData.RealData ));
					gThickData.ControlOk = 0;
					gThickData.FocusNum  = 0;
					TimePid.OutMax =  gThickProf.ShareSet.ThickFlow * 33;
					TimePid.OutMin = -1 * TimePid.OutMax ;

					SetPID = gThickData.SetData[0];

					//				for (uTIndex = 0; uTIndex < 100; uTIndex++)
					//				{
					//					gThickData.SetData[uTIndex] = gTempData[uTIndex];
					//				}
					TimeCtrlStep = 40;
					break;

				case 40:                                   /* Time mode profile */
					if(ABS(vHydDT2Set.y) > vSetLimit || ABS(vHydDT2Act.y) > vActLimit)
					{
						//    TimePid.KiGain = 0;
					}

					// Call function

					//				for (uTIndex = 0; uTIndex < 100; uTIndex++)
					//				{
					//					gThickData.SetData[uTIndex] = gTempData[uTIndex];
					//				}

					TimeCurveData(&gThickData);

					SetPID = gThickData.SetPID;

					gThickData.CurrentTime = gThickData.Counter/5;

					if(1 == gThickData.ControlOk)
					{
						gThickData.CurrentTime = 0;
						gThickData.ControlOk = 0;
						TimeCtrlStep = 50;
					}
					break;

				case 50:
					gThickData.StartServoPos = TimePid.Act;
					gThickData.Counter  = 0;
					gThickData.FocusNum = 0;
					TimePid.OutMax =  gThickProf.ShareSet.SealFlow * 33;
					TimePid.OutMin = -1 * TimePid.OutMax ;

					ContolEndTime = 100;
					gThickIO.Out.ControlEnd = 1;

					SetPID = TimePid.Act;

					if(0 == gThickProf.FunOption.SealMode)
					{
						SealValue = gThickData.SetData[0];
					}
					else
					{
						SealValue = gThickData.SealPos;
					}

					TimeCtrlStep = 60;
					break;

				case 60:
					gThickData.Counter++;                    /* 封口时间 */
					if((SealValue - gThickData.StartServoPos != 0) && (gThickData.SealGapDly != 0))
					{
						SetPID = (short)(gThickData.StartServoPos + ( SealValue - gThickData.StartServoPos)
							* gThickData.Counter / gThickData.SealGapDly);
					}
					else
					{
						SetPID = SealValue;
					}

					if(gThickData.Counter >= gThickData.SealGapDly)
					{
						gThickData.Counter = 0;
						TimeCtrlStep = 100;
					}
					break;

				case 100:
					if(0 == gThickProf.FunOption.SealMode)
					{
						SetPID = gThickData.SetData[0];
					}
					else
					{
						SetPID = gThickData.SealPos;
					}
					break;

				/*  ----------------- Seal gap -------------------- */
				case 110:
					gThickData.StartServoPos = TimePid.Act;
					gThickData.Counter  = 0;
					gThickData.FocusNum = 0;
					TimePid.OutMax =  gThickProf.ShareSet.SealFlow * 33;
					TimePid.OutMin = -1 * TimePid.OutMax ;

					SetPID = TimePid.Act;
					SealValue = gThickData.SealPos;

					TimeCtrlStep = 120;
					break;

				case 120:
					gThickData.Counter++;           /* 封口时间 */
					if((SealValue - gThickData.StartServoPos != 0) && (gThickData.SealGapDly != 0))
					{
						SetPID = (short)(gThickData.StartServoPos + ( SealValue - gThickData.StartServoPos)
							* gThickData.Counter / gThickData.SealGapDly);
					}
					else
					{
						SetPID = SealValue;
					}

					if(gThickData.Counter >= gThickData.SealGapDly)
					{
						gThickData.Counter = 0;
						TimeCtrlStep = 130;
					}
					break;

				case 130:
					gThickData.Counter++;
					if(gThickData.Counter > 2000)
					{
						gThickData.Counter = 0;
						TimeCtrlStep = 140;
					}
					break;

				case 140:
					gThickData.StartServoPos = TimePid.Act;
					gThickData.Counter  = 0;
					gThickData.FocusNum = 0;
					TimePid.OutMax =  gThickProf.ShareSet.SealFlow * 33;
					TimePid.OutMin = -1 * TimePid.OutMax ;

					SetPID = TimePid.Act;

					if(0 == gThickProf.FunOption.SealMode)
					{
						SealValue = gThickData.SetData[0];
					}
					else
					{
						SealValue = gThickData.SealPos;
					}

					TimeCtrlStep = 150;
					break;

				case 150:
					gThickData.Counter++;           /* 封口时间 */
					if((SealValue - gThickData.StartServoPos != 0) && (gThickData.SealGapDly != 0))
					{
						SetPID = (short)(gThickData.StartServoPos + ( SealValue - gThickData.StartServoPos)
							* gThickData.Counter / gThickData.SealGapDly);
					}
					else
					{
						SetPID = SealValue;
					}

					if(gThickData.Counter >= gThickData.SealGapDly)
					{
						gThickData.Counter = 0;
						TimeCtrlStep = 200;
					}
					break;

				case 200:
					if(0 == gThickProf.FunOption.SealMode)
					{
						SetPID = gThickData.SetData[0];
					}
					else
					{
						SetPID = gThickData.SealPos;
					}
					break;

				default:
					SetPID = gServoLinear.Current;
					break;

			}/* switch(TimeCtrlStep) */

			if(0 == gThickIO.In.Purge && 0 == PurgeOld)
			{
				RampSet.Set = SetPID;
			}
			else if(gThickIO.In.Purge != PurgeOld)
			{
				RampSet.Once = 0;
				RampSet.Set  = gServoLinear.Current;
			}
			else if(1 == gThickIO.In.Purge && 1 == PurgeOld)
			{
				RampSet.Set = gThickData.PurgePos;
			}

			/* Call function  */
			HydRampCos(&RampSet);

			if(0 == gThickIO.In.Purge && 0 == PurgeOld)
			{
				TimePid.Set = SetPID;
			}
			else
			{
				TimePid.Set = RampSet.Out;
			}

			PIDCtrl(&TimePid);

			SetValue = TimePid.Set;
			ServeOut = TimePid.Out + TimePid.RepairOut;

			if(40 == TimeCtrlStep)
			{
				gControlInfo.CurrentPoint = gThickData.FocusNum;
				if(1 ==gThickProf. IsMarker[gThickData.FocusNum])
				{
					MarkerTime = 125;
				}
			}
			else
			{
				gControlInfo.CurrentPoint = 0;
			}

			AccuCtrlStep = 100;
		}
		else  /* if(0 == gThickProf.FunOption.IsAccu) */  /* 位置式 */
		{
			switch(AccuCtrlStep)
			{
				case 10:
					gThickData.Counter = 0;
					gThickData.StartServoPos = AccuPid.Act;
					AccuPid.OutMax =  gThickProf.ShareSet.StartFlow * 33;
					AccuPid.OutMin = -1 * AccuPid.OutMax ;

					RampSet.Once = 0;
					SetPID = AccuPid.Act;

					AccuCtrlStep = 20;
					break;

				case 20:                                 /* 开口延迟 */
					gThickData.Counter++;

					if((gThickData.SetData[0] - gThickData.StartServoPos != 0) && (gThickData.AccuOpenDly != 0))
					{
						SetPID = (short)(gThickData.StartServoPos + (gThickData.SetData[0] - gThickData.StartServoPos)
							* gThickData.Counter / gThickData.AccuOpenDly );
					}
					else
					{
						SetPID = gThickData.SetData[0];
					}
					if(gThickData.Counter >= gThickData.AccuOpenDly )
					{
						gThickData.Counter = 0;
						AccuCtrlStep = 30;
					}
					break;

				case 30:
					gThickData.CurrentTime = 0;
					gThickData.ControlOk   = 0;
					gThickData.FocusNum    = 0;
					memset(gThickData.RealData ,0,sizeof(gThickData.RealData ));
					memset(gThickData.InitLock ,1,sizeof(gThickData.InitLock));
					AccuPid.OutMax =  gThickProf.ShareSet.ThickFlow * 33;
					AccuPid.OutMin = -1 * AccuPid.OutMax ;

					SetPID = gThickData.SetData[0];

					gThickData.CurrentPos = gAccuLinear.Current - gThickData.Offset;

					AccuCtrlStep = 40;
					break;

				case 40:                                 /* 位置式控制 */
					if(ABS(vHydDT2Set.y) > vSetLimit || ABS(vHydDT2Act.y) > vActLimit)
					{
						AccuPid.KiGain = 0;
					}

					gThickData.CurrentPos = gAccuLinear.Current - gThickData.Offset;

					/* call function  */
					AccuCurveData(&gThickData);

					SetPID = gThickData.SetPID;

					if(1 == gThickData.ControlOk)
					{
						gThickData.ControlOk = 0;
						gThickData.Counter = 0;
						AccuCtrlStep = 50;
					}
					break;

				case 50:
					if(0 == gTKauto.Status)
					{
						gThickData.StartServoPos = AccuPid.Act;
					}
					else
					{
						gThickData.StartServoPos = gThickData.SetData[99];
					}
					gThickData.FocusNum = 0;
					gThickData.Offset = 0;

					SetPID = AccuPid.Act;

					AccuCtrlStep = 60;
					break;

				case 60:
					SetPID = gThickData.StartServoPos;
					break;

				case 100:
					gThickData.StartServoPos = AccuPid.Act;
					gThickData.Counter = 0;
					AccuPid.OutMax =  gThickProf.ShareSet.SealFlow * 33;
					AccuPid.OutMin = -1 * AccuPid.OutMax ;

					RampSet.Once = 0;
					SetPID = AccuPid.Act;

					AccuCtrlStep = 110;
					break;

				case 110:                                /* 封口时间 */
					gThickData.Counter++;

					if((gThickData.SealPos - gThickData.StartServoPos != 0) && (gThickData.SealGapDly != 0))
					{
						SetPID = (short)(gThickData.StartServoPos + (gThickData.SealPos - gThickData.StartServoPos)
							* gThickData.Counter / gThickData.SealGapDly);
					}
					else
					{
						SetPID = gThickData.SealPos;
					}

					if(gThickData.Counter >= gThickData.SealGapDly)
					{
						gThickData.Counter = 0;
						AccuCtrlStep = 120;
					}
					break;

				case 120:
					SetPID = gThickData.SealPos;
					AccuCtrlStep = 200;
					break;

				case 200:
					SetPID = gThickData.SealPos;
					break;

				default:
					SetPID = gServoLinear.Current;
					break;
			}/* switch(AccuCtrlStep) */

			if(0 == gThickIO.In.Purge && 0 == PurgeOld)
			{
				RampSet.Set = SetPID;
			}
			else if(gThickIO.In.Purge != PurgeOld)
			{
				RampSet.Once = 0;
				RampSet.Set  = gServoLinear.Current;
			}
			else if(1 == gThickIO.In.Purge && 1 == PurgeOld)
			{
				RampSet.Set = gThickData.PurgePos;
			}

			HydRampCos(&RampSet);

			if(0 == gThickIO.In.Purge && 0 == PurgeOld)
			{
				AccuPid.Set = SetPID;
			}
			else
			{
				AccuPid.Set = RampSet.Out;
			}

			PIDCtrl(&AccuPid);

			SetValue = AccuPid.Set;
			ServeOut = AccuPid.Out + AccuPid.RepairOut;

			if(40 == AccuCtrlStep)
			{
				gControlInfo.CurrentPoint = gThickData.FocusNum;
				if(1 == gThickProf.IsMarker[gThickData.FocusNum])
				{
					MarkerTime = 125;
				}
			}
			else
			{
				gControlInfo.CurrentPoint = 0;
			}

			TimeCtrlStep = 50;
		}/* else if(0 == gThickProf.FunOption.IsAccu) */

		if((gThickData.ServoMax - gThickData.ServoMin) != 0)
		{
			if(0 == gThickProf.FunOption.IsZeroDn)
			{
				gThickIO.SetPercent = (SetValue - gThickData.ServoMin            )* 100.0 /(gThickData.ServoMax - gThickData.ServoMin);
				gThickIO.ActPercent = (gServoLinear.Current - gThickData.ServoMin)* 100.0 /(gThickData.ServoMax - gThickData.ServoMin);
			}
			else
			{
				gThickIO.SetPercent = (gThickData.ServoMax - SetValue            )* 100.0 /(gThickData.ServoMax - gThickData.ServoMin);
				gThickIO.ActPercent = (gThickData.ServoMax - gServoLinear.Current)* 100.0 /(gThickData.ServoMax - gThickData.ServoMin);
			}
		}
		else
		{
			gThickIO.SetPercent = 0.0;
			gThickIO.ActPercent = 0.0;
		}

		cmdAutoCalibrate = 0;
		CalibrateStep = 0;
		SetGapValue = gServoLinear.Current;

		/* keep mode */
		SetGapPercent = gThickIO.SetPercent;
		bCalibPosMode = 0;
	}
	else     /* 调校状态 */
	{
		SetPID = gServoLinear.Current;

		gThickIO.SetPercent = 0.0;

		gThickIO.In.Stop     = 0;
		gThickIO.In.SealGap  = 0;

		ServeSetValue = gServoLinear.Current;
		/* thickness time  */
		if(1 == gThickIO.In.StartThick)
		{
			gThickIO.In.StartThick = 0;
			CycleTimeCount = gThickData.CycleTimes + 1;
		}

		if(CycleTimeCount > 0)CycleTimeCount--;
		gThickData.CurrentTime = (gThickData.CycleTimes - CycleTimeCount) / 5;
		if(1 == CycleTimeCount)gThickIO.Out.ControlEnd = 1;
		if(0 == CycleTimeCount)gThickData.CurrentTime = 0;

		if(gThickProf.TimSet.CycleTime != 0)
		{
			gThickData.FocusNum = gThickData.CurrentTime * 10.0/gThickProf.TimSet.CycleTime;
		}

		/*  判断是否手动校调和自动校调  */
		if(cmdServoUp != 0              || cmdServoDn != 0    || cmdAutoCalibrate != 0       || CalibrateStep != 0 ||
			0 == gMachineOut.ParisonPump || gServoLinear.Current < gThickData.ServoMin - 1635 || gServoLinear.Current > gThickData.ServoMax + 1635)
		{
			bCalibPosMode = 0;
		}

		if(0 == bCalibPosMode)
		{
			if(0 == gThickProf.FunOption.IsAutoCalibrate)  /* 手动调校 */
			{
				if(1 == cmdServoUp)
				{
					ServeOut = -gServoLinear.ManualSpeed ;
				}

				if(1 == cmdServoDn)
				{
					ServeOut = gServoLinear.ManualSpeed;
				}

				if((0 == cmdServoUp) &&(0 == cmdServoDn))
				{
					ServeOut = 0;
					bCalibPosMode = 1;
					SetGapPercent = gThickIO.ActPercent;
				}
				CalibrateStep = 0;
			}
			else                                           /* 自动调校 */
			{
				if(1 == cmdAutoCalibrate)
				{
					cmdAutoCalibrate = 0;
					if(gServoLinear.AutoSpeed > 0 && 0 == CalibrateStep)
					{
						CalibrateStep = 10;
					}
				}

				/* step machine control  */
				switch(CalibrateStep)
				{
					case 0:
						ServeOut = 0;
						break;

					case 10:
						gServoLinear.Status = 2;
						TimeCount = 0;
						CurrentInput = gServoLinear.Current;
						LastInput    = gServoLinear.Current;
						CalibrateStep = 20;
						break;

					case 20:
						ServeOut = -gServoLinear.AutoSpeed;
						TimeCount++;

						if( 0 == (TimeCount % 1000))
						{
							CurrentInput = gServoLinear.Current;
							if( (CurrentInput - LastInput) > -100 && (CurrentInput - LastInput) < 100 )
							{
								CalibrateStep = 30;
							}
							LastInput = CurrentInput;
						}
						break;

					case 30:
						gServoLinear.ZeroPos = gServoLinear.Current;
						ServeOut  = 0;
						TimeCount = 0;
						CurrentInput = gServoLinear.Current;
						LastInput    = gServoLinear.Current;
						CalibrateStep = 40;
						break;

					case 40:
						ServeOut = gServoLinear.AutoSpeed;
						TimeCount++;

						if( 0 == (TimeCount % 1000))
						{
							CurrentInput = gServoLinear.Current;
							if( (CurrentInput - LastInput) > -100 && (CurrentInput - LastInput) < 100 )
							{
								CalibrateStep = 50;
							}
							LastInput = CurrentInput;
						}
						break;

					case 50:
						gServoLinear.MaxPos = gServoLinear.Current;
						ServeOut  = 0;
						TimeCount = 0;
						CalibrateStep = 60;
						break;

					case 60:
						gServoLinear.Status = gServoLinear.IsReady;
						gRecipeOperate.OnceSave = 1;
						CalibrateStep = 0;
						break;

					default:
						break;
				}/* switch(CalibrateStep) */
			} /* 自动调校 */

			if((gThickData.ServoMax - gThickData.ServoMin) != 0)
			{
				if(0 == gThickProf.FunOption.IsZeroDn)
				{
					gThickIO.ActPercent = (gServoLinear.Current - gThickData.ServoMin)* 100.0 /(gThickData.ServoMax - gThickData.ServoMin);
				}
				else
				{
					gThickIO.ActPercent = (gThickData.ServoMax - gServoLinear.Current)* 100.0 /(gThickData.ServoMax - gThickData.ServoMin);
				}
			}
			else
			{
				gThickIO.ActPercent = 0.0;
			}
			SetGapValue = gServoLinear.Current;
		}
		else                    /*  keep mode  */
		{
			if((gThickData.ServoMax - gThickData.ServoMin) != 0)
			{
				if(0 == gThickProf.FunOption.IsZeroDn)
				{
					SetGapValue = gThickData.ServoMin + (gThickData.ServoMax - gThickData.ServoMin)* SetGapPercent/100.0;
					gThickIO.ActPercent = (gServoLinear.Current - gThickData.ServoMin)* 100.0 /(gThickData.ServoMax - gThickData.ServoMin);
				}
				else
				{
					SetGapValue = gThickData.ServoMax - (gThickData.ServoMax - gThickData.ServoMin)* SetGapPercent/100.0;
					gThickIO.ActPercent = (gThickData.ServoMax - gServoLinear.Current)* 100.0 /(gThickData.ServoMax - gThickData.ServoMin);
				}
			}
			else
			{
				gThickIO.ActPercent = 0.0;
			}

			CalibPid.Set = (INT)RampCalibSet.Out;
			if(CalibPid.e0 > 100 || CalibPid.e0 < -100)CalibPid.KiGain = 0;
			PIDCtrl(&CalibPid);
			ServeOut = CalibPid.Out + CalibPid.RepairOut;
		}
		TimeCtrlStep = 50;
		AccuCtrlStep = 100;
		gThickIO.Out.MarkPulse  = 0;
	} /* else 调校状态 */

	RampCalibSet.Set = SetGapValue;
	HydSCurveRamp(&RampCalibSet);

	if(1 == bSetCalibPos)
	{
		bSetCalibPos = 0;
		bCalibPosMode = 1;
		CalibPid.Yi = 0;
	}

	if(bCalibPosModeOld != bCalibPosMode)
	{
		CalibPid.Yi = 0;
	}
	bCalibPosModeOld = bCalibPosMode;

	gControlInfo.CurrentGapSet = SetGapValue;
	gControlInfo.CurrentGapSetPercent = gThickIO.SetPercent;

	gControlInfo.CurrentGapPercent = gThickIO.ActPercent;

	if(MarkerTime > 0)
	{
		MarkerTime--;
		gThickIO.Out.MarkPulse  = 1;
	}
	else
	{
		gThickIO.Out.MarkPulse  = 0;
	}

	if(StartTime > 0)
	{
		StartTime --;
		gThickIO.Out.Start = 1;
	}
	else
	{
		gThickIO.Out.Start = 0;
	}

	if(ContolEndTime > 0)
	{
		ContolEndTime--;
		gThickIO.Out.End  = 1;
	}
	else
	{
		gThickIO.Out.End  = 0;
	}

	Wave = -1 * Wave;

	if(gServoLinear.Current < 32767     && gServoLinear.Current > 0 &&
		1 == gThickProf.FunOption.Servo  && 1 == gMachineOut.ParisonPump)
	{
		gThickIO.ServoOut = (short)( ServeOut + Wave * TimePid.Wave);
	}
	else
	{
		gThickIO.ServoOut = 0;
	}

	gMachineOut.StartThick = gThickIO.Out.Start;
	PurgeOld = gThickIO.In.Purge;

}/*  end of cycle  */
```

#### parison.var
```iecst
VAR
	tTask : REAL := 0.0;
	RTInfo_Task : RTInfo := (0);
	TimeCtrlStep : INT;
	AccuCtrlStep : INT;
	CalibrateStep : INT;
	cmdAutoCalibrate : BOOL;
	cmdServoUp : BOOL;
	cmdServoDn : BOOL;
	SetValue : INT;
	ServeSetValue : INT;
	CycleTimeCount : UDINT;
	Wave : INT;
	SetPID : DINT;
	ServeOut : DINT;
	TimeCount : UDINT;
	CurrentInput : INT;
	LastInput : INT;
	MarkerTime : UDINT;
	ContolEndTime : UDINT;
	SealValue : INT;
	rSetPercent : REAL;
	rActPercent : REAL;
	StartTime : UDINT;
	CalibPid : Thick_PID_typ;
	bSetCalibPos : USINT;
	bCalibPosMode : USINT;
	bCalibPosModeOld : USINT;
	PurgeOld : USINT;
	SetGapValue : REAL;
	RampCalibSet : HydSCurveRamp;
	RampSet : HydRampCos;
	vHydDT2Set : HydDT2;
	vSetLimit : REAL;
	vHydDT2Act : HydDT2;
	vActLimit : REAL;
	SetGapPercent : REAL;
END_VAR
(*Insert your comment here.*)
VAR
	uTIndex : UINT;
END_VAR
```

- thick.c (not readable text: treated as protected, skipped)

- thick.h (reference to Logical/GlobalIncludes/thick.h)

### Package Logical/screen - HMI Setting and password

### screen.var - Global variables
```iecst
(********************************************************************
 * COPYRIGHT --
 ********************************************************************
 * Package: screen
 * File: screen.var
 * Author: lij
 * Created: December 19, 2013
 ********************************************************************
 * Variables of package screen
 ********************************************************************)
VAR RETAIN
	OldRTCTime : RTCtime_typ;
END_VAR
```

### Program Logical/screen/keyled (ANSIC, version 1.00.0) - key led control

#### keyled.c
```c
/********************************************************************
 * COPYRIGHT --  B&R China
 ********************************************************************
 * Program: panel
 * File: panel.c
 * Author: lijianjun
 * Created: March 06, 2013
 ********************************************************************
 * Implementation of program panel --- display led control
 ********************************************************************/

#include <bur/plctypes.h>

#ifdef _DEFAULT_INCLUDES
#include <AsDefault.h>
#endif

#include "defines.h"
#include "edge.h"
#include "keyap2100.h"
//#include "keyap880.h"
#include "pic_id.h"

/**************************************************************************************
     	        		I N I T U P  O F   T H E   T A S K
**************************************************************************************/
_INIT void init ( void )
{
} /* end of _INIT */

 /*************************************************************************************
        				C Y C L I C   P A R T   O F   T H E   T A S K
**************************************************************************************/

_CYCLIC void cyclic ( void )
{
	/* ------------------ VK key and Real key ------------------ */

	for(index=0;index<32;index++)  /*  5AP880.1505 KEY L1 - L12 F1 - F16 R1 - R12 */
	{
		//ipis0218
		if ((gPanelObj.PasswordLevel >=1))
		{
			if ((1==gMachineIn.OilPumpOk_DI && 1==gMachineInfo.OilPumpDelayDone)  && (0 == btnTesetPQ))
			{
				if( index <= 19 /*&& (1== gMachineInfo.Manual)*/)
				{
					if(  1 == gPanelObj.RKeyMatric[index] && 1 == gPanelObj.KeyMatric[index] )
					{
						index_Main = index;
						Lock_Flag = 1;
					}
					else if(  0 == gPanelObj.RKeyMatric[index_Main] && 1 == Lock_Flag )
					{
						index_Main = 0;
						Lock_Flag = 0;
					}

					if( 0 == Lock_Flag )
					{
						gPanelObj.KeyMatric[index] = gPanelObj.RKeyMatric[index] | gPanelObj.VKeyMatric[index] | gPanelObj.MKeyMatric[index];
					}
				}
				else
				{
					gPanelObj.KeyMatric[index] = gPanelObj.RKeyMatric[index] | gPanelObj.VKeyMatric[index] | gPanelObj.MKeyMatric[index];
				}
			}
		}
		else
		{
			if (gPanelObj.PasswordLevel < 1)
			{
				if (EDGEPOS(gPanelObj.RKeyMatric[index],RKeyMatric[index]) || EDGEPOS(gPanelObj.VKeyMatric[index],RKeyMatric[index]) )
				{
					gImply.PsdLevel1=1;
				}
			}
		}

		//		if ((0==gMachineIn.OilPumpOk_DI || 0==gMachineInfo.OilPumpDelayDone))
		//		{
		//			if (EDGEPOS(gPanelObj.RKeyMatric[index],RKeyMatric[index]) || EDGEPOS(gPanelObj.VKeyMatric[index],RKeyMatric[index]) )
		//			{
		//				gImply.OilPumpNotOn=1;
		//			}
		//		}

		//		if(EDGEPOS(gPanelObj.KeyMatric[index],PKeyMatric[index]) )
		//		{
		//			if(1 == gMachineInfo.Manual || 1 == gMachineInfo.Calib )
		//			{
		//				if ( 1 == gMachineInfo.IsImply ) gMachineOut.ImplyBuzzer  = 1;
		//			}
		//
		//		}
		//
		//		if(EDGENEG(gPanelObj.KeyMatric[index],NKeyMatric[index]) )
		//		{
		//			gMachineOut.ImplyBuzzer  = 0;
		//		}

	}

	//		if ((1==gMachineIn.OilPumpOk_DI && 1==gMachineInfo.OilPumpDelayDone)  && (0 == btnTesetPQ))
	//		{
	//			for(index=0;index<22;index++)  /*  5AP880.1505 KEY L1 - L12 F1 - F16 R1 - R12 */
	//			{
	//				gPanelObj.KeyMatric[index] = gPanelObj.RKeyMatric[index] | gPanelObj.VKeyMatric[index] | gPanelObj.MKeyMatric[index];
	//
	//			}
	//		}

	for(index=32;index<400;index++)  /*  5AP880.1505 KEY L1 - L12 F1 - F16 R1 - R12 */
	{
		gPanelObj.KeyMatric[index] = gPanelObj.RKeyMatric[index] | gPanelObj.VKeyMatric[index] | gPanelObj.MKeyMatric[index];
	}

	//	if ((0==gMachineIn.OilPumpOk_DI || 0==gMachineInfo.OilPumpDelayDone))
	//	{
	//
	//		for(index=0;index<22;index++)  /*  5AP880.1505 KEY L1 - L12 F1 - F16 R1 - R12 */
	//		{
	//			if (EDGEPOS(gPanelObj.RKeyMatric[index],RKeyMatric[index]) )
	//			{
	//				gImply.OilPumpNotOn=1;
	//			}
	//		}
	//	}

	//	for(index=0;index<400;index++)  /*  5AP880.1505 KEY L1 - L12 F1 - F16 R1 - R12 */
	//   {
	//      gPanelObj.KeyMatric[index] = gPanelObj.RKeyMatric[index] | gPanelObj.VKeyMatric[index] | gPanelObj.MKeyMatric[index];
	//   }

	//	for(index=100;index<200;index++)
	//	{
	//		gPanelObj.KeyMatric[index] = gPanelObj.RKeyMatric[index] | gPanelObj.VKeyMatric[index] | gPanelObj.MKeyMatric[index];
	//	}
	//
	//	for(index=276;index<296;index++)  /*  5AC800.EX2-01  number key and arrow key  */
	//	{
	//		gPanelObj.KeyMatric[index - OFFSET_EX2_01] = gPanelObj.RKeyMatric[index] | gPanelObj.VKeyMatric[index] | gPanelObj.MKeyMatric[index];
	//	}

	/* ------------------ ActInfo ------------------ */
	ActInfo.ClampCls    = LMold.ActInfo.ClampCls | RMold.ActInfo.ClampCls;
	ActInfo.ClampOpn    = LMold.ActInfo.ClampOpn | RMold.ActInfo.ClampOpn;

	ActInfo.CarriageFw  = LMold.ActInfo.CarriageFw | RMold.ActInfo.CarriageFw;
	ActInfo.CarriageBw  = LMold.ActInfo.CarriageBw | RMold.ActInfo.CarriageBw;

	ActInfo.BlowPinDn   = LMold.ActInfo.BlowPinDn  | RMold.ActInfo.BlowPinDn;
	ActInfo.BlowPinUp   = LMold.ActInfo.BlowPinUp  | RMold.ActInfo.BlowPinUp;

	ActInfo.LowBlow 	= gMachineOut.LMold.LowBlow  | gMachineOut.RMold.LowBlow;
	ActInfo.HighBlow 	= gMachineOut.LMold.HighBlow  | gMachineOut.RMold.HighBlow;

	ActInfo.ExtrLiftUp 	= LMold.ActInfo.ExtrLiftUp | RMold.ActInfo.ExtrLiftUp;
	ActInfo.ExtrLiftDn 	= LMold.ActInfo.ExtrLiftDn | RMold.ActInfo.ExtrLiftDn;

	ActInfo.Cutter      = LMold.ActInfo.Cutter | RMold.ActInfo.Cutter;
	ActInfo.InnerPin 	= LMold.ActInfo.InnerPin   | RMold.ActInfo.InnerPin;
	ActInfo.PullBottom 	= LMold.ActInfo.PullBottom | RMold.ActInfo.PullBottom;
	ActInfo.CoolPinDn   = LMold.ValveOut.CoolPinDn | RMold.ValveOut.CoolPinDn;
	ActInfo.CoolPinBlow	= LMold.ValveOut.CoolPinBlow | RMold.ValveOut.CoolPinBlow;
	ActInfo.CoolPin2Dn  = LMold.ValveOut.CoolPin2Dn | RMold.ValveOut.CoolPin2Dn;
	ActInfo.CoolPin2Blow= LMold.ValveOut.CoolPin2Blow | RMold.ValveOut.CoolPin2Blow;
	ActInfo.CoolPin3Dn  = LMold.ValveOut.CoolPin3Dn | RMold.ValveOut.CoolPin3Dn;
	ActInfo.CoolPin3Blow= LMold.ValveOut.CoolPin3Blow | RMold.ValveOut.CoolPin3Blow;
	ActInfo.BlowDeflash = LMold.ActInfo.BlowDeflash  | RMold.ActInfo.BlowDeflash;
	ActInfo.CoolDeflash = LMold.ActInfo.CoolDeflash  | RMold.ActInfo.CoolDeflash;
	ActInfo.SubMoldOpn	= LMold.ActInfo.SubMoldOpn | RMold.ActInfo.SubMoldOpn;
	ActInfo.SubMoldCls	= LMold.ActInfo.SubMoldCls | RMold.ActInfo.SubMoldCls;
	ActInfo.PinPartFw	= LMold.ActInfo.PinPartFw | RMold.ActInfo.PinPartFw;
	ActInfo.PinPartBw	= LMold.ActInfo.PinPartBw | RMold.ActInfo.PinPartBw;
	ActInfo.ScrewFw		= LMold.ActInfo.ScrewFw   | RMold.ActInfo.ScrewFw;
	ActInfo.ScrewBw		= LMold.ActInfo.ScrewBw   | RMold.ActInfo.ScrewBw;
	ActInfo.RobotFw		= LMold.ValveOut.RobotFw  | RMold.ValveOut.RobotFw | ( ACTUATOR_PNEU != gMachineFix.MoldR.RobotTransfer.eActuatorType && (LMold.ActInfo.RobotFw| RMold.ActInfo.RobotFw));
	ActInfo.RobotBw		= LMold.ValveOut.RobotBw  | RMold.ValveOut.RobotBw | ( ACTUATOR_PNEU != gMachineFix.MoldR.RobotTransfer.eActuatorType && (LMold.ActInfo.RobotBw| RMold.ActInfo.RobotBw));
	ActInfo.RobotCls	= LMold.ValveOut.RobotCls | RMold.ValveOut.RobotCls;
	ActInfo.RobotUp		= LMold.ValveOut.RobotUp  | RMold.ValveOut.RobotUp;
	ActInfo.RobotDn		= LMold.ValveOut.RobotDn  | RMold.ValveOut.RobotDn;
	ActInfo.CutNeck		= LMold.ValveOut.CutNeck    | RMold.ValveOut.CutNeck;
	ActInfo.CutNeckCls	= LMold.ValveOut.CutNeckCls | RMold.ValveOut.CutNeckCls;
	ActInfo.SupportAir	= gMachineOut.SupportAir_1 || gMachineOut.SupportAir_TimeVersion ;
	ActInfo.TopDeflashFw = LMold.ValveOut.TopDeflashFw  | RMold.ValveOut.TopDeflashFw;
	ActInfo.TopDeflashBw = LMold.ValveOut.TopDeflashBw  | RMold.ValveOut.TopDeflashBw;
	ActInfo.BottomDeflashFw = LMold.ValveOut.BottomDeflashFw  | RMold.ValveOut.BottomDeflashFw;
	ActInfo.BottomDeflashBw = LMold.ValveOut.BottomDeflashBw  | RMold.ValveOut.BottomDeflashBw;
	ActInfo.PullBottom 	= LMold.ValveOut.PullBottom  | RMold.ValveOut.PullBottom;
	ActInfo.HookPinFw  = LMold.ValveOut.HookPinFw | RMold.ValveOut.HookPinFw;

	/*  5AP880.1505 KEY L1 - L12 */
	gPanelObj.LedMatric[S$KEYMATRIX_MAIN_PUMP] = gMachineOut.OilPump;
		gPanelObj.LedMatric[S$KEYMATRIX_PARISON_PUMP] = gMachineOut.ParisonPump;

		gPanelObj.LedMatric[S$KEYMATRIX_HEAT_POWER] = gMachineOut.HeatPower;

		//	gPanelObj.LedMatric[S$KEYMATRIX_EXTRUDER_A] = gMachineIn.ExtrA_OnOff;
		//	gPanelObj.LedMatric[S$KEYMATRIX_EXTRUDER_B] = gMachineIn.ExtrB_OnOff;

		//	gPanelObj.LedMatric[S$KEYMATRIX_EXTRUDER_A_PLK] = gExtruderACtrl.InverterStatus.bSwitchOn;/*Albert*/
		//	gPanelObj.LedMatric[S$KEYMATRIX_EXTRUDER_B_PLK] = gExtruderBCtrl.InverterStatus.bSwitchOn;/*Albert*/
		//	gPanelObj.LedMatric[S$KEYMATRIX_EXTRUDER_C_PLK] = gExtruderCCtrl.InverterStatus.bSwitchOn;/*Albert*/
		//	gPanelObj.LedMatric[S$KEYMATRIX_VISU_EXTRUDER_PLK] = gExtruderVCtrl.InverterStatus.bSwitchOn;/*Albert*/

		//		gPanelObj.LedMatric[S$KEYMATRIX_EXTRUDER_A_PLK] = gMachineOut.ExtrA_Enable;/*ipis*/
		//		gPanelObj.LedMatric[S$KEYMATRIX_EXTRUDER_B_PLK] = gMachineOut.ExtrB_Enable;/*ipis*/
		//		gPanelObj.LedMatric[S$KEYMATRIX_EXTRUDER_C_PLK] = gMachineOut.ExtrC_Enable;/*ipis*/
		//		gPanelObj.LedMatric[S$KEYMATRIX_VISU_EXTRUDER_PLK] = gMachineOut.ExtrV_Enable;/*ipis*/

		/* for ABB inveter ------------------------------------------------*/
		gPanelObj.LedMatric[S$KEYMATRIX_EXTRUDER_A_ABB] = gMachineOut.ExtrA_On;
		gPanelObj.LedMatric[S$KEYMATRIX_EXTRUDER_B_ABB] = gMachineOut.ExtrB_On;
		gPanelObj.LedMatric[S$KEYMATRIX_EXTRUDER_C_ABB] = gMachineOut.ExtrC_On;
		gPanelObj.LedMatric[S$KEYMATRIX_EXTRUDER_D_ABB] = gMachineOut.ExtrD_On;
		if(1 == gMachineFix.ExtruderD.LinkWithMode && 1 == gMachineFix.ExtruderVisu.LinkWithMode)
	{
		gPanelObj.LedMatric[S$KEYMATRIX_EXTRUDER_D_ABB] = gMachineOut.ExtrD_On || gMachineOut.ExtrVisu_On;
			}
	else
	{
		gPanelObj.LedMatric[S$KEYMATRIX_EXTRUDER_D_ABB] = gMachineOut.ExtrD_On;
			}
	/*---------------------------------------------------------------------------*/

	gPanelObj.LedMatric[S$KEYMATRIX_MODE_CALIB] = gMachineInfo.Calib;
		gPanelObj.LedMatric[S$KEYMATRIX_MODE_MANUAL]= gMachineInfo.Manual;
		gPanelObj.LedMatric[S$KEYMATRIX_MODE_AUTO]  = gMachineInfo.Auto;
		gPanelObj.LedMatric[S$KEYMATRIX_AUTO_RESET] = gMachineInfo.MachineReset;

		gPanelObj.LedMatric[S$KEYMATRIX_AUTO_STOP] = (2 == gMachineInfo.LedAutoStop) ;/*Albert*/

		gPanelObj.LedMatric[S$KEYMATRIX_CUTTER_FW]   = ActInfo.Cutter;
		if( ACTUATOR_ELECTRIC  == gMachineFix.ExtrLift.eActuatorType )
	{
		gPanelObj.LedMatric[S$KEYMATRIX_EXTRUDER_UP] = ActInfo.ExtrLiftUp;
			gPanelObj.LedMatric[S$KEYMATRIX_EXTRUDER_DN] = ActInfo.ExtrLiftDn;
			}
	else
	{
		gPanelObj.LedMatric[S$KEYMATRIX_EXTRUDER_UP] = ActInfo.ExtrLiftUp||ActInfo.ExtrLiftDn;
			}

	if (1==gMacOption.Station) //Right ipis0128
	{
		gPanelObj.LedMatric[S$KEYMATRIX_CARRIAGE_UP] = ActInfo.CarriageFw;
			gPanelObj.LedMatric[S$KEYMATRIX_CARRIAGE_DN] = ActInfo.CarriageBw;
			}
	if (0==gMacOption.Station) //Left ipis0128
	{
		gPanelObj.LedMatric[S$KEYMATRIX_CARRIAGE_UP] = ActInfo.CarriageBw;
			gPanelObj.LedMatric[S$KEYMATRIX_CARRIAGE_DN] = ActInfo.CarriageFw;
			}
	if (2==gMacOption.Station) //Right ipis0129
	{
		gPanelObj.LedMatric[S$KEYMATRIX_CARRIAGE_UP] = RMold.ActInfo.CarriageFw ||LMold.ActInfo.CarriageBw;
			gPanelObj.LedMatric[S$KEYMATRIX_CARRIAGE_DN] = RMold.ActInfo.CarriageFw ||LMold.ActInfo.CarriageFw ;
			}

	gPanelObj.LedMatric[S$KEYMATRIX_CLAMP_OPN ]  = ActInfo.ClampOpn;
		gPanelObj.LedMatric[S$KEYMATRIX_CLAMP_CLS]   = ActInfo.ClampCls;
		gPanelObj.LedMatric[S$KEYMATRIX_BLOWPIN_UP]  = ActInfo.BlowPinUp;
		gPanelObj.LedMatric[S$KEYMATRIX_BLOWPIN_DN]  = ActInfo.BlowPinDn;

		gPanelObj.LedMatric[S$KEYMATRIX_PLATE_UP] = gMachineOut.PlateUp;
		gPanelObj.LedMatric[S$KEYMATRIX_PLATE_DN] = gMachineOut.PlateDn;
		gPanelObj.LedMatric[S$KEYMATRIX_TOP_DEFLASH_FW] = ActInfo.TopDeflashFw;
		//	gPanelObj.LedMatric[S$KEYMATRIX_BOT_DEFLASH_FW] = ActInfo.BottomDeflash;
		//	gPanelObj.LedMatric[S$KEYMATRIX_BOT_DEFLASH_FW] = ActInfo.BottomDeflashFw;
		gPanelObj.LedMatric[S$KEYMATRIX_TOP_DEFLASH_BW] = ActInfo.TopDeflashBw;
		//	gPanelObj.LedMatric[S$KEYMATRIX_BOT_DEFLASH_BW] = ActInfo.BottomDeflashBw;
		gPanelObj.LedMatric[S$KEYMATRIX_PULL_BOTTOM_FW] = ActInfo.PullBottom;

		gPanelObj.LedMatric[S$KEYMATRIX_ROBOT_FW]  = ActInfo.RobotFw;
		gPanelObj.LedMatric[S$KEYMATRIX_ROBOT_BW]  = ActInfo.RobotBw;
		//	gPanelObj.LedMatric[S$KEYMATRIX_ROBOT_FWBW] =ActInfo.RobotFw ||ActInfo.RobotBw ;
		gPanelObj.LedMatric[S$KEYMATRIX_ROBOT_CLS] = ActInfo.RobotCls;
		gPanelObj.LedMatric[S$KEYMATRIX_BLOW]      = ActInfo.HighBlow;
		gPanelObj.LedMatric[S$KEYMATRIX_SUPPORT]   = ActInfo.SupportAir;
		gPanelObj.LedMatric[S$KEYMATRIX_COOL_DEFLASH]   = ActInfo.CoolDeflash;
		gPanelObj.LedMatric[S$KEYMATRIX_CUT_NECK]   = ActInfo.CutNeck;

		gPanelObj.LedMatric[S$KEYMATRIX_LUBRICATION] = gMachineOut.Lubricate;
		gPanelObj.LedMatric[S$KEYMATRIX_DRY_CYCLE] = gMachineInfo.bDryCycle = gMacOption.bDryCycle;
		//	gPanelObj.LedMatric[S$KEYMATRIX_PRODUCTAUX_CLS] = LMold.ValveOut.ProductAuxClamp  | RMold.ValveOut.ProductAuxClamp;

		gPanelObj.LedMatric[S$KEYMATRIX_COOL_DN] = ActInfo.CoolPinDn;
		gPanelObj.LedMatric[S$KEYMATRIX_COOL_BLOW] = ActInfo.CoolPinBlow;

		gPanelObj.LedMatric[S$KEYMATRIX_COOL2_DN] = ActInfo.CoolPin2Dn;
		gPanelObj.LedMatric[S$KEYMATRIX_COOL2_BLOW] = ActInfo.CoolPin2Blow;

		gPanelObj.LedMatric[S$KEYMATRIX_COOL3_DN] = ActInfo.CoolPin3Dn;
		gPanelObj.LedMatric[S$KEYMATRIX_COOL3_BLOW] = ActInfo.CoolPin3Blow;

		/*Albert Led status of PIC_FAST_SETTING*/

		/*IO DI*/
		//	if(gPanelObj.GetPicture == PIC_IO_DI_1)
		//	{
		//		gPanelObj.LedMatric[S$PAGE_MONITOR] = 1;
		//	}
		//	else
		//	{
		//		gPanelObj.LedMatric[S$PAGE_MONITOR] = 0;
		//	}
		//
		//	/*Temperature*/
		//	if(gPanelObj.GetPicture == PIC_TEMP_ALL)
		//	{
		//		gPanelObj.LedMatric[S$PAGE_TEMP_ALL] = 1;
		//	}
		//	else
		//	{
		//		gPanelObj.LedMatric[S$PAGE_TEMP_ALL] = 0;
		//	}
		//
		//	/*Extruder Speed */
		//	if(gPanelObj.GetPicture == PIC_SPEED)
		//	{
		//		gPanelObj.LedMatric[S$PAGE_EXTRUDER] = 1;
		//	}
		//	else
		//	{
		//		gPanelObj.LedMatric[S$PAGE_EXTRUDER] = 0;
		//	}

		/*------------------------------------------------------------*/

		gHardWare.XP0101Led_1[1]  = gMachineOut.LMold.BlowPinDnHold  | gMachineOut.RMold.BlowPinDnHold;;
	if ((1==LMold.Option.SubMold&& 0==LMold.Option.BottomSubMold) || (1==RMold.Option.SubMold&& 0==RMold.Option.BottomSubMold))    //ipis0128 topsubmold
	{
		gHardWare.XP0101Led_1[5]  = ActInfo.SubMoldCls;
		gHardWare.XP0101Led_1[9]  = ActInfo.SubMoldOpn;
	}
	if ((1==LMold.Option.BottomSubMold&&0==LMold.Option.SubMold) || (1==RMold.Option.BottomSubMold&&0==RMold.Option.SubMold)) //ipis0128 BottomSubMold
	{
		gHardWare.XP0101Led_1[5]  = ActInfo.SubMoldOpn;
		gHardWare.XP0101Led_1[9]  = ActInfo.SubMoldCls;
	}

	gHardWare.XP0101Led_1[13] = gMachineOut.PlateUp;;
	gHardWare.XP0101Led_1[17] = gMachineOut.PlateDn;

	if (6600==RMold.Plate.Step || 6600==LMold.Plate.Step) //ipis0802
	{
		gHardWare.XP0101Led_1[21] = 0;
	}
	else
	{
		gHardWare.XP0101Led_1[21] = gMachineOut.PlateFw;

	}

	gHardWare.XP0101Led_1[25] = gMachineOut.PlateBw;

	if(gPanelObj.GetPicture == PIC_FAST_SETTING)
	{
		gHardWare.XP0101Led_1[29] = 1;
	}
	else
	{
		gHardWare.XP0101Led_1[29] = 0;
	}

} /* end of _CYCLIC */
```

#### keyled.var
```iecst
VAR
	index : UINT;
	ActInfo : Act_Info_typ;
	RKeyMatric : ARRAY[0..MAX_KEY_COUNT] OF USINT;
	PKeyMatric : ARRAY[0..MAX_KEY_COUNT] OF USINT;
	NKeyMatric : ARRAY[0..MAX_KEY_COUNT] OF USINT;
	Lock_Flag : USINT;
	index_Main : USINT;
END_VAR
```

### Program Logical/screen/hmiset (ANSIC, version 1.00.0) - HMI set

#### hmiset.c
```c
/********************************************************************
 * COPYRIGHT --  B&R China
 ********************************************************************
 * Program: hmiset
 * File: hmiset.c
 * Author: lijianjun
 * Created: March 06, 2013
 ********************************************************************
 * Implementation of program hmiset --- HMI setting parameter control
 ********************************************************************/

#include <bur/plctypes.h>

#ifdef _DEFAULT_INCLUDES
	#include <AsDefault.h>
#endif

#include <string.h>
/*********************************************************************************
** 							    defines                     			                 **
*********************************************************************************/
#define S$STEP_SETUP 		   10
#define S$STEP_IDLE 			   20
#define S$STEP_SETCONTRAST 	30
#define S$STEP_SETBRIGHTNESS 	40

#define S$STEP_INIT 			    0
#define S$STEP_GET_TIME 	  100
#define S$STEP_SET_TIME 	  200
/********************************************************************************
****	        		I N I T U P  O F   T H E   T A S K 		 		              ****
********************************************************************************/
_INIT void hmiset_Init(void)
{
	hmiStep  = S$STEP_SETUP;
   hmiTimeStep = S$STEP_INIT;

   strcpy(gPanelObj.VisualName, "visu15");
}
/*********************************************************************************
***    C Y C L I C   P A R T   O F   T H E   T A S K  			              ****
*********************************************************************************/
_CYCLIC void hmiset_Cyclic(void)
{

	BackLightTime = hmiBackLightTime_Min *60;

    STRING NumName[5];

	/*  contrast and brigfhtness set in hmi */
	switch (hmiStep)
	{
		case S$STEP_SETUP:
			gPanelObj.vcHandle = VA_Setup(1, gPanelObj.VisualName);

			if (gPanelObj.vcHandle != 0)
			{
				if (!VA_Saccess(1, gPanelObj.vcHandle))
				{
					Contrast = VA_GetContrast(1,gPanelObj.vcHandle);
					contrast_old = Contrast;

					VA_GetBrightness(1,gPanelObj.vcHandle,(UDINT)&Brightness);
					brightness_old = Brightness;

					VA_Srelease(1, gPanelObj.vcHandle);
				}
				hmiStep = S$STEP_IDLE;
			}
		break;

		case S$STEP_IDLE:		/* wait for changes in contrast/brightness setting */
			/* Limit Values */
			if (Contrast   > 100)Contrast   = 100;
			if (Brightness > 100)Brightness = 100;

			if (Contrast != contrast_old)
			{
				contrast_old = Contrast ;
				hmiStep = S$STEP_SETCONTRAST;
			}
			else if (Brightness != brightness_old)
			{
				brightness_old = Brightness ;
				hmiStep = S$STEP_SETBRIGHTNESS;
			}
		break;

		case S$STEP_SETCONTRAST:	/* set new contrast value */
			if (!VA_Saccess(1, gPanelObj.vcHandle))
			{
				VA_SetContrast(1, gPanelObj.vcHandle, Contrast);
				VA_Srelease(1, gPanelObj.vcHandle);
			}
			hmiStep = S$STEP_IDLE;
		break;

		case S$STEP_SETBRIGHTNESS:	/* set new brightness value */
			if (!VA_Saccess(1, gPanelObj.vcHandle))
			{
				VA_SetBrightness(1, gPanelObj.vcHandle, Brightness);
				VA_Srelease(1, gPanelObj.vcHandle);
			}
			hmiStep = S$STEP_IDLE;
		break;
	}/* switch (hmiStep) */

    /* -------------------------- system time set in HMI -------------------------- */
    switch (hmiTimeStep)
    {
        case S$STEP_INIT:				   /*  Init start   */
            RTC_gettime(&GetRTCTime);
            SetRTCTime = GetRTCTime;

            /*  定时停机  */
            if(!OldRTCTime.year)    	/* 第一次下载  */
            {
               OldRTCTime = GetRTCTime;
					gMachineWorkDays = 0;
               gMachineStopDays = 0;
            }
            else
            {
            	if(GetRTCTime.year >= OldRTCTime.year)     /*  battery keep */
               {
						gMachineWorkDays = gMachineWorkDays + ((GetRTCTime.year - OldRTCTime.year)* 12 + GetRTCTime.month - OldRTCTime.month) * 30
						                      + GetRTCTime.day - OldRTCTime.day;
                  gMachineStopDays = gMachineStopDays + ((GetRTCTime.year - OldRTCTime.year)* 12 + GetRTCTime.month - OldRTCTime.month) * 30
                        + GetRTCTime.day - OldRTCTime.day;
               }
               OldRTCTime = GetRTCTime;
            }/* if(!OldRTCTime.year) */

            hmiTimeStep = S$STEP_GET_TIME;
            break;
        case S$STEP_GET_TIME :
            if((SetRTCTime.hour   != GetRTCTime.hour)     ||
               (SetRTCTime.minute != GetRTCTime.minute)   ||
               (SetRTCTime.second != GetRTCTime.second)   ||
               (SetRTCTime.month  != GetRTCTime.month)    ||
               (SetRTCTime.day    != GetRTCTime.day )     ||
               (SetRTCTime.year   != GetRTCTime.year))
            {
                hmiTimeStep = S$STEP_SET_TIME ;
            }
            else
            {
                RTC_gettime(&GetRTCTime);
                SetRTCTime = GetRTCTime;

                if(GetRTCTime.day != GetRTCTime.day )
                {
						 gMachineWorkDays++;
                   gMachineStopDays++;
                }

                OldRTCTime = GetRTCTime;

                strcpy(gPanelObj.Password4,"");
                strcpy(CurrentTime,"");
                strcpy(Time,"");
                itoa((long)(GetRTCTime.year ),(unsigned long)NumName);
                strcat(Time,NumName);

                strcat(gPanelObj.Password4,NumName);

                strcat(Time,"-");
                if(GetRTCTime.month < 10)
                {
                    strcat(Time,"0");
                }
                itoa((long)(GetRTCTime.month ),(unsigned long)NumName);
                strcat(Time,NumName);
                strcat(Time,"-");

                if(GetRTCTime.day < 10)
                {
                    strcat(Time,"0");
                }
                itoa((long)(GetRTCTime.day ),(unsigned long)NumName);
                strcat(Time,NumName);

                strcat(CurrentTime,Time);

                strcat(CurrentTime," ");

                if(GetRTCTime.hour < 10)
                {
                    strcat(CurrentTime,"0");
                }
                itoa((long)(GetRTCTime.hour ),(unsigned long)NumName);
                strcat(CurrentTime,NumName);

                strcat(CurrentTime,":");
                if(GetRTCTime.minute < 10)
                {
                    strcat(CurrentTime,"0");
                }
                itoa((long)(GetRTCTime.minute ),(unsigned long)NumName);
                strcat(CurrentTime,NumName);

                strcpy(gPanelObj.CurrentTime,CurrentTime);

                strcat(gPanelObj.CurrentTime,":");
                if(GetRTCTime.second < 10)
                {
                    strcat(gPanelObj.CurrentTime,"0");
                }
                itoa((long)(GetRTCTime.second ),(unsigned long)NumName);
                strcat(gPanelObj.CurrentTime,NumName);

                strcpy(gPanelObj.PasswordHigh,"2016");

                itoa((long)(GetRTCTime.day%10),(unsigned long)NumName);
                strcat(gPanelObj.PasswordHigh,NumName);

                itoa((long)(GetRTCTime.hour%10),(unsigned long)NumName);
                strcat(gPanelObj.PasswordHigh,NumName);

                itoa((long)(GetRTCTime.minute/10),(unsigned long)NumName);
                strcat(gPanelObj.PasswordHigh,NumName);

                itoa((long)(GetRTCTime.hour%10),(unsigned long)NumName);
                strcat(gPanelObj.Password4,NumName);

                itoa((long)(GetRTCTime.minute%10),(unsigned long)NumName);
                strcat(gPanelObj.Password4,NumName);
            }
            break;
        case S$STEP_SET_TIME :

            RTC_settime(&SetRTCTime);

            if((SetRTCTime.day   != OldRTCTime.day  ) ||
               (SetRTCTime.month != OldRTCTime.month) ||
               (SetRTCTime.year  != OldRTCTime.year ))
            {
                gMachineStopDays++;
            }
            OldRTCTime = SetRTCTime;
            GetRTCTime = SetRTCTime;

            hmiTimeStep = S$STEP_INIT;
            break;
    }

}/* end of cycle */
/* ----------------------------------------------------------------------------- */
```

#### hmiset.var
```iecst
VAR
	hmiStep : UINT;
	Contrast : UDINT;
	BackLightTime : UINT;
END_VAR
VAR RETAIN
	hmiBackLightTime_Min : UINT;
END_VAR
VAR
	contrast_old : UINT;
	Brightness : UDINT;
	brightness_old : UINT;
END_VAR
(*time setting *)
VAR
	hmiTimeStep : UINT;
	Time : STRING[11];
	CurrentTime : STRING[18];
	GetRTCTime : RTCtime_typ := (0);
	SetRTCTime : RTCtime_typ := (0);
END_VAR
```

### Program Logical/screen/scrshot (ANSIC, version 1.00.0) - copy screen to usb disk
